KUKA KRL program: MyProgram_040().src

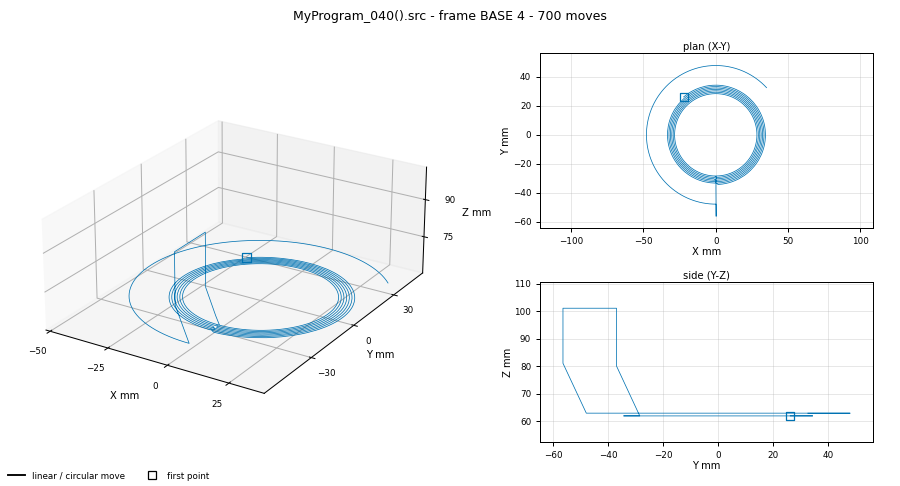
[picture p0: tool path of MyProgram_040().src in frame BASE 4, 700 of 700 moves have a stored position in this frame; points joined in program order, loops and branches not executed]
&ACCESS RVP
&REL 1
&PARAM TEMPLATE = C:\KRC\Roboter\Template\vorgabe
&PARAM EDITMASK = *
DEF MyProgram_040()
; ---- Setting reference (Base) ----
$BASE = BASE_DATA[4]

; --------------------------
; ---- Setting tool (TCP) ----
$TOOL = TOOL_DATA[3]
; --------------------------

$VEL.CP = VEL_APROX_PRINT
Startdeposition()
$VEL.CP = VEL_PRINT
LIN {X -22.2135,Y 26.2071,Z 62,A 121.4467,B 24.8242,C -3.0577,E1 24.9,E2 -758.4485} C_DIS
LIN {X -19.0591,Y 28.5827,Z 62,A 115.8795,B 24.8216,C -3.0802,E1 24.9125,E2 -752.9155} C_DIS
LIN {X -17.4873,Y 29.5709,Z 62,A 112.412,B 24.8214,C -3.0822,E1 24.9208,E2 -749.4421} C_DIS
LIN {X -15.634,Y 30.5912,Z 62,A 108.9316,B 24.8207,C -3.0885,E1 24.9293,E2 -745.967} C_DIS
LIN {X -13.2901,Y 31.6799,Z 62,A 103.9982,B 24.8207,C -3.0886,E1 24.942,E2 -741.0221} C_DIS
LIN {X -10.8187,Y 32.6071,Z 62,A 99.9719,B 24.8196,C -3.0977,E1 24.9525,E2 -737.0096} C_DIS
LIN {X -8.4739,Y 33.2931,Z 62,A 96.4896,B 24.8184,C -3.1079,E1 24.9618,E2 -733.5462} C_DIS
LIN {X -7.1425,Y 33.6045,Z 62,A 93.5529,B 24.819,C -3.1031,E1 24.9699,E2 -730.5943} C_DIS
LIN {X -4.6609,Y 34.0375,Z 62,A 89.325,B 24.8187,C -3.1056,E1 24.9816,E2 -726.3687} C_DIS
LIN {X -2.445,Y 34.2678,Z 62,A 85.3655,B 24.8187,C -3.1047,E1 24.9926,E2 -722.4051} C_DIS
LIN {X 0.711,Y 34.3473,Z 62,A 80.7474,B 24.8178,C -3.1129,E1 25.0054,E2 -717.8067} C_DIS
LIN {X 2.5788,Y 34.2575,Z 62,A 77.4409,B 24.8181,C -3.1108,E1 25.0146,E2 -714.4965} C_DIS
LIN {X 4.6969,Y 34.0324,Z 62,A 74.1424,B 24.8178,C -3.1131,E1 25.0238,E2 -711.2059} C_DIS
LIN {X 6.978,Y 33.6386,Z 62,A 70.5125,B 24.8176,C -3.1144,E1 25.0337,E2 -707.583} C_DIS
LIN {X 8.415,Y 33.3079,Z 62,A 67.7146,B 24.8183,C -3.109,E1 25.0413,E2 -704.7764} C_DIS
LIN {X 10.1674,Y 32.8156,Z 62,A 64.7507,B 24.8184,C -3.1078,E1 25.0493,E2 -701.8147} C_DIS
LIN {X 12.5471,Y 31.9815,Z 62,A 59.7382,B 24.82,C -3.0942,E1 25.0625,E2 -696.7805} C_DIS
LIN {X 14.5005,Y 31.1445,Z 62,A 56.4765,B 24.82,C -3.0937,E1 25.0707,E2 -693.5258} C_DIS
LIN {X 16.8742,Y 29.9253,Z 62,A 52.3714,B 24.8202,C -3.0922,E1 25.0808,E2 -689.4289} C_DIS
LIN {X 19.1187,Y 28.5434,Z 62,A 47.4262,B 24.8218,C -3.0785,E1 25.0924,E2 -684.4673} C_DIS
LIN {X 20.7359,Y 27.3913,Z 62,A 43.8567,B 24.8229,C -3.0695,E1 25.1004,E2 -680.8892} C_DIS
LIN {X 23.4463,Y 25.1103,Z 62,A 38.3676,B 24.8236,C -3.0636,E1 25.1119,E2 -675.408} C_DIS
LIN {X 25.8911,Y 22.5808,Z 62,A 32.7892,B 24.8246,C -3.0549,E1 25.1224,E2 -669.8333} C_DIS
LIN {X 27.3559,Y 20.7829,Z 62,A 29.4122,B 24.8248,C -3.0525,E1 25.1283,E2 -666.4667} C_DIS
LIN {X 28.1113,Y 19.7485,Z 62,A 27.0275,B 24.8258,C -3.0439,E1 25.1322,E2 -664.0731} C_DIS
LIN {X 29.1969,Y 18.1051,Z 62,A 23.9145,B 24.8265,C -3.038,E1 25.1369,E2 -660.9619} C_DIS
LIN {X 30.04,Y 16.6688,Z 62,A 21.2563,B 24.8271,C -3.0324,E1 25.1405,E2 -658.3041} C_DIS
LIN {X 30.6921,Y 15.435,Z 62,A 18.4558,B 24.8286,C -3.0195,E1 25.1441,E2 -655.4879} C_DIS
LIN {X 31.6221,Y 13.4275,Z 62,A 14.5033,B 24.8302,C -3.0056,E1 25.1486,E2 -651.524} C_DIS
LIN {X 32.6254,Y 10.7638,Z 62,A 10.1437,B 24.8311,C -2.9974,E1 25.1526,E2 -647.1695} C_DIS
LIN {X 33.1185,Y 9.1348,Z 62,A 7.3906,B 24.8319,C -2.9902,E1 25.1547,E2 -644.4151} C_DIS
LIN {X 33.5819,Y 7.246,Z 62,A 4.3845,B 24.8327,C -2.9839,E1 25.1566,E2 -641.4115} C_DIS
LIN {X 33.9043,Y 5.5446,Z 62,A 1.3815,B 24.8338,C -2.9735,E1 25.158,E2 -638.4014} C_DIS
LIN {X 34.175,Y 3.5099,Z 62,A -2.0165,B 24.835,C -2.9633,E1 25.1592,E2 -634.9993} C_DIS
LIN {X 34.3202,Y 1.5388,Z 62,A -5.2617,B 24.836,C -2.9538,E1 25.1597,E2 -631.7509} C_DIS
LIN {X 34.3541,Y 0.1987,Z 62,A -7.6725,B 24.8371,C -2.9442,E1 25.1597,E2 -629.3319} C_DIS
LIN {X 34.309,Y -1.7741,Z 62,A -10.9313,B 24.8382,C -2.9344,E1 25.1594,E2 -626.0691} C_DIS
LIN {X 34.0961,Y -4.2062,Z 62,A -14.637,B 24.839,C -2.9269,E1 25.1584,E2 -622.3678} C_DIS
LIN {X 33.8382,Y -5.9366,Z 62,A -17.6519,B 24.8402,C -2.9164,E1 25.157,E2 -619.3456} C_DIS
LIN {X 33.4085,Y -8.0083,Z 62,A -21.3611,B 24.8417,C -2.9028,E1 25.1547,E2 -615.6259} C_DIS
LIN {X 32.8832,Y -9.9486,Z 62,A -24.8083,B 24.8429,C -2.8912,E1 25.152,E2 -612.1708} C_DIS
LIN {X 32.0411,Y -12.3943,Z 62,A -28.5367,B 24.8434,C -2.8866,E1 25.1485,E2 -608.4525} C_DIS
LIN {X 31.434,Y -13.8624,Z 62,A -32.1813,B 24.8458,C -2.8645,E1 25.1444,E2 -604.7755} C_DIS
LIN {X 29.7344,Y -17.2082,Z 62,A -37.2411,B 24.8459,C -2.8637,E1 25.1379,E2 -599.7404} C_DIS
LIN {X 28.506,Y -19.1745,Z 62,A -42.1252,B 24.8486,C -2.8387,E1 25.1304,E2 -594.8215} C_DIS
LIN {X 26.7916,Y -21.5054,Z 62,A -47.2958,B 24.8505,C -2.8213,E1 25.1215,E2 -589.6341} C_DIS
LIN {X 23.923,Y -24.6562,Z 62,A -53.4408,B 24.8509,C -2.8174,E1 25.1097,E2 -583.5064} C_DIS
LIN {X 21.6339,Y -26.6874,Z 62,A -59.2704,B 24.8531,C -2.7963,E1 25.0972,E2 -577.6496} C_DIS
LIN {X 19.7191,Y -28.1322,Z 62,A -63.5381,B 24.8543,C -2.7848,E1 25.0875,E2 -573.3694} C_DIS
LIN {X 15.9551,Y -30.425,Z 62,A -69.5933,B 24.8539,C -2.7889,E1 25.0729,E2 -567.3422} C_DIS
LIN {X 13.6297,Y -31.5353,Z 62,A -74.5651,B 24.8555,C -2.7737,E1 25.0602,E2 -562.3468} C_DIS
LIN {X 11.1987,Y -32.4787,Z 62,A -78.4482,B 24.8555,C -2.774,E1 25.05,E2 -558.4725} C_DIS
LIN {X 9.155,Y -33.1128,Z 62,A -82.0156,B 24.8559,C -2.7701,E1 25.0405,E2 -554.9019} C_DIS
LIN {X 6.777,Y -33.6799,Z 62,A -86.4571,B 24.8567,C -2.762,E1 25.0283,E2 -550.447} C_DIS
LIN {X 4.3543,Y -34.0777,Z 62,A -89.9455,B 24.8562,C -2.7665,E1 25.0187,E2 -546.9726} C_DIS
LIN {X 1.6468,Y -34.3153,Z 62,A -95.2543,B 24.8574,C -2.7554,E1 25.0039,E2 -541.6397} C_DIS
LIN {X 1.6468,Y -34.3153,Z 62,A -95.2543,B 24.8574,C -2.7554,E1 25.0039,E2 -541.6397} C_DIS
Enddeposition()
LIN {X 0.1829,Y -33.3699,Z 62,A -96.4469,B 24.8542,C -2.7864,E1 25.0008,E2 -540.5209} C_DIS
Startdeposition()
$VEL.CP = VEL_PRINT
LIN {X 1.4228,Y -33.3445,Z 62,A -93.237,B 24.8528,C -2.7995,E1 25.0098,E2 -543.7614} C_DIS
LIN {X 3.8682,Y -33.1501,Z 62,A -89.4536,B 24.8531,C -2.7966,E1 25.0203,E2 -547.5356} C_DIS
LIN {X 6.4667,Y -32.7422,Z 62,A -84.1849,B 24.8518,C -2.8092,E1 25.0348,E2 -552.8286} C_DIS
LIN {X 8.6813,Y -32.2262,Z 62,A -80.8923,B 24.8521,C -2.8055,E1 25.0437,E2 -556.1074} C_DIS
LIN {X 10.7356,Y -31.6013,Z 62,A -76.8197,B 24.8512,C -2.8147,E1 25.0546,E2 -560.1942} C_DIS
LIN {X 13.1904,Y -30.658,Z 62,A -72.1573,B 24.8503,C -2.8228,E1 25.0667,E2 -564.8654} C_DIS
LIN {X 15.1524,Y -29.7371,Z 62,A -69.1058,B 24.8506,C -2.82,E1 25.0743,E2 -567.9021} C_DIS
LIN {X 16.9825,Y -28.7313,Z 62,A -64.8683,B 24.849,C -2.8349,E1 25.0846,E2 -572.1622} C_DIS
LIN {X 18.9767,Y -27.4551,Z 62,A -61.3792,B 24.849,C -2.8349,E1 25.0927,E2 -575.6399} C_DIS
LIN {X 21.2128,Y -25.7669,Z 62,A -55.8058,B 24.8468,C -2.8555,E1 25.105,E2 -581.2413} C_DIS
LIN {X 22.9178,Y -24.2625,Z 62,A -51.6212,B 24.8454,C -2.8684,E1 25.1135,E2 -585.4392} C_DIS
LIN {X 25.8376,Y -21.1265,Z 62,A -45.1587,B 24.8448,C -2.8741,E1 25.1255,E2 -591.8865} C_DIS
LIN {X 27.6388,Y -18.708,Z 62,A -39.68,B 24.8428,C -2.8922,E1 25.1344,E2 -597.3815} C_DIS
LIN {X 29.0319,Y -16.4634,Z 62,A -35.1975,B 24.8415,C -2.9042,E1 25.1408,E2 -601.8693} C_DIS
LIN {X 30.4402,Y -13.6854,Z 62,A -30.0332,B 24.8401,C -2.9171,E1 25.147,E2 -607.0365} C_DIS
LIN {X 31.2986,Y -11.588,Z 62,A -26.4051,B 24.8392,C -2.925,E1 25.1507,E2 -610.6631} C_DIS
LIN {X 31.92,Y -9.7482,Z 62,A -22.6045,B 24.8374,C -2.9419,E1 25.1539,E2 -614.4821} C_DIS
LIN {X 32.7265,Y -6.5492,Z 62,A -17.7367,B 24.8367,C -2.9479,E1 25.157,E2 -619.3359} C_DIS
LIN {X 32.9464,Y -5.3344,Z 62,A -14.5179,B 24.8342,C -2.9705,E1 25.1584,E2 -622.5894} C_DIS
LIN {X 33.3383,Y -1.5702,Z 62,A -9.092,B 24.8336,C -2.9753,E1 25.1597,E2 -627.9943} C_DIS
LIN {X 33.375,Y 0.0538,Z 62,A -6.2185,B 24.8325,C -2.9852,E1 25.1597,E2 -630.8742} C_DIS
LIN {X 33.3259,Y 1.8094,Z 62,A -3.2231,B 24.8315,C -2.9943,E1 25.1594,E2 -633.8734} C_DIS
LIN {X 33.2052,Y 3.364,Z 62,A -0.7318,B 24.8308,C -2.9999,E1 25.1588,E2 -636.3632} C_DIS
LIN {X 33.0427,Y 4.6979,Z 62,A 1.6423,B 24.8299,C -3.008,E1 25.1579,E2 -638.7425} C_DIS
LIN {X 32.7913,Y 6.2155,Z 62,A 4.524,B 24.8286,C -3.0195,E1 25.1565,E2 -641.6345} C_DIS
LIN {X 32.2699,Y 8.5188,Z 62,A 8.4206,B 24.8275,C -3.0294,E1 25.1539,E2 -645.5319} C_DIS
LIN {X 31.633,Y 10.6416,Z 62,A 12.4439,B 24.8259,C -3.0436,E1 25.1505,E2 -649.566} C_DIS
LIN {X 30.8002,Y 12.855,Z 62,A 16.3295,B 24.8248,C -3.0526,E1 25.1465,E2 -653.4515} C_DIS
LIN {X 29.4508,Y 15.7026,Z 62,A 22.0288,B 24.8227,C -3.0713,E1 25.1394,E2 -659.1647} C_DIS
LIN {X 28.245,Y 17.7799,Z 62,A 25.5541,B 24.8224,C -3.0736,E1 25.1343,E2 -662.6774} C_DIS
LIN {X 27.4035,Y 19.051,Z 62,A 28.1395,B 24.8217,C -3.0796,E1 25.1303,E2 -665.2643} C_DIS
LIN {X 26.5171,Y 20.267,Z 62,A 30.6298,B 24.8211,C -3.0845,E1 25.1261,E2 -667.7543} C_DIS
LIN {X 25.6944,Y 21.3,Z 62,A 32.9585,B 24.8204,C -3.0906,E1 25.122,E2 -670.0865} C_DIS
LIN {X 24.7958,Y 22.3399,Z 62,A 36.0169,B 24.8187,C -3.1052,E1 25.1163,E2 -673.1659} C_DIS
LIN {X 22.7484,Y 24.4218,Z 62,A 40.7734,B 24.8179,C -3.1119,E1 25.1067,E2 -677.9187} C_DIS
LIN {X 20.6615,Y 26.2106,Z 62,A 45.0491,B 24.8176,C -3.1148,E1 25.0976,E2 -682.1848} C_DIS
LIN {X 19.1465,Y 27.337,Z 62,A 48.6346,B 24.8164,C -3.1247,E1 25.0894,E2 -685.7811} C_DIS
LIN {X 17.0397,Y 28.6975,Z 62,A 52.5144,B 24.8164,C -3.1256,E1 25.0803,E2 -689.6509} C_DIS
LIN {X 15.4263,Y 29.5963,Z 62,A 55.9993,B 24.8154,C -3.1337,E1 25.0717,E2 -693.145} C_DIS
LIN {X 13.597,Y 30.48,Z 62,A 59.7045,B 24.8146,C -3.1404,E1 25.0623,E2 -696.8566} C_DIS
LIN {X 11.4187,Y 31.3607,Z 62,A 63.0646,B 24.8151,C -3.136,E1 25.0536,E2 -700.199} C_DIS
LIN {X 10.1374,Y 31.7985,Z 62,A 65.3843,B 24.8149,C -3.1378,E1 25.0474,E2 -702.5184} C_DIS
LIN {X 8.378,Y 32.3064,Z 62,A 68.9747,B 24.814,C -3.1451,E1 25.0377,E2 -706.1203} C_DIS
LIN {X 6.1328,Y 32.8069,Z 62,A 72.6936,B 24.8141,C -3.1441,E1 25.0276,E2 -709.8324} C_DIS
LIN {X 4.5023,Y 33.0705,Z 62,A 75.876,B 24.8136,C -3.1488,E1 25.0187,E2 -713.0232} C_DIS
LIN {X 1.7164,Y 33.3311,Z 62,A 81.564,B 24.8124,C -3.1589,E1 25.0028,E2 -718.7328} C_DIS
LIN {X -2.4774,Y 33.2834,Z 62,A 87.3966,B 24.8144,C -3.1417,E1 24.9867,E2 -724.5252} C_DIS
LIN {X -3.8653,Y 33.1504,Z 62,A 90.0327,B 24.8142,C -3.143,E1 24.9793,E2 -727.1661} C_DIS
LIN {X -5.6675,Y 32.8906,Z 62,A 93.1198,B 24.8146,C -3.1405,E1 24.9708,E2 -730.25} C_DIS
LIN {X -7.3587,Y 32.554,Z 62,A 96.5725,B 24.8142,C -3.1431,E1 24.9614,E2 -733.7131} C_DIS
LIN {X -9.9318,Y 31.8625,Z 62,A 100.6041,B 24.8155,C -3.1328,E1 24.9506,E2 -737.7267} C_DIS
LIN {X -12.8323,Y 30.8096,Z 62,A 106.8089,B 24.8152,C -3.1348,E1 24.9344,E2 -743.9496} C_DIS
LIN {X -15.1762,Y 29.725,Z 62,A 110.2748,B 24.8171,C -3.1186,E1 24.9258,E2 -747.3857} C_DIS
LIN {X -16.7138,Y 28.8886,Z 62,A 113.5931,B 24.8174,C -3.1165,E1 24.9177,E2 -750.7086} C_DIS
LIN {X -18.3349,Y 27.8877,Z 62,A 117.4181,B 24.8174,C -3.1156,E1 24.9087,E2 -754.5439} C_DIS
LIN {X -21.0824,Y 25.8722,Z 62,A 122.2135,B 24.82,C -3.094,E1 24.8981,E2 -759.305} C_DIS
LIN {X -22.0783,Y 25.0293,Z 62,A 126.1085,B 24.8189,C -3.104,E1 24.8899,E2 -763.2393} C_DIS
LIN {X -25.5295,Y 21.4982,Z 62,A 134.6867,B 24.8212,C -3.0841,E1 24.8738,E2 -771.808} C_DIS
LIN {X -28.2172,Y 17.8241,Z 62,A 141.0536,B 24.825,C -3.0507,E1 24.8638,E2 -778.1262} C_DIS
LIN {X -28.9128,Y 16.6716,Z 62,A 143.5735,B 24.8256,C -3.046,E1 24.8602,E2 -780.648} C_DIS
LIN {X -29.7714,Y 15.0848,Z 62,A 146.4195,B 24.8268,C -3.0351,E1 24.8565,E2 -783.4829} C_DIS
LIN {X -30.2718,Y 14.0538,Z 62,A 149.4607,B 24.8265,C -3.0383,E1 24.8529,E2 -786.5483} C_DIS
LIN {X -31.6705,Y 10.5303,Z 62,A 154.8201,B 24.8298,C -3.0093,E1 24.8477,E2 -791.8686} C_DIS
LIN {X -32.3711,Y 8.1254,Z 62,A 160.5197,B 24.83,C -3.0075,E1 24.8435,E2 -797.5971} C_DIS
LIN {X -32.8497,Y 5.8982,Z 62,A 164.193,B 24.8316,C -2.9934,E1 24.8416,E2 -801.2584} C_DIS
LIN {X -33.2606,Y 2.7623,Z 62,A 169.0956,B 24.834,C -2.9722,E1 24.8401,E2 -806.1394} C_DIS
LIN {X -33.3722,Y 0.439,Z 62,A 173.4965,B 24.835,C -2.963,E1 24.8398,E2 -810.5449} C_DIS
LIN {X -33.3243,Y -1.8394,Z 62,A 177.3186,B 24.8364,C -2.9501,E1 24.8402,E2 -814.359} C_DIS
LIN {X -33.1418,Y -3.9387,Z 62,A -179.5093,B 24.8381,C -2.9353,E1 24.8411,E2 -817.5147} C_DIS
LIN {X -32.9043,Y -5.5852,Z 62,A -176.45,B 24.8389,C -2.9282,E1 24.8425,E2 -820.5753} C_DIS
LIN {X -32.5254,Y -7.4827,Z 62,A -173.0592,B 24.8399,C -2.9188,E1 24.8445,E2 -823.9635} C_DIS
LIN {X -31.9568,Y -9.6266,Z 62,A -169.2266,B 24.8411,C -2.9078,E1 24.8474,E2 -827.7919} C_DIS
LIN {X -31.1362,Y -12.0183,Z 62,A -164.5872,B 24.8422,C -2.8979,E1 24.8518,E2 -832.4338} C_DIS
LIN {X -30.1887,Y -14.2317,Z 62,A -160.582,B 24.8436,C -2.8854,E1 24.8564,E2 -836.4311} C_DIS
LIN {X -29.4655,Y -15.6747,Z 62,A -157.8731,B 24.8444,C -2.8774,E1 24.8599,E2 -839.1354} C_DIS
LIN {X -28.295,Y -17.6999,Z 62,A -153.9787,B 24.8457,C -2.8661,E1 24.8655,E2 -843.0228} C_DIS
LIN {X -27.374,Y -19.0935,Z 62,A -151.2935,B 24.8466,C -2.8574,E1 24.8697,E2 -845.7005} C_DIS
LIN {X -26.456,Y -20.3464,Z 62,A -148.4701,B 24.8471,C -2.8525,E1 24.8744,E2 -848.5257} C_DIS
LIN {X -25.3348,Y -21.7268,Z 62,A -145.3707,B 24.8478,C -2.846,E1 24.88,E2 -851.6239} C_DIS
LIN {X -24.0752,Y -23.1145,Z 62,A -142.0378,B 24.8485,C -2.8402,E1 24.8863,E2 -854.9575} C_DIS
LIN {X -22.8098,Y -24.3641,Z 62,A -139.1432,B 24.8493,C -2.8326,E1 24.8921,E2 -857.8459} C_DIS
LIN {X -21.4959,Y -25.5315,Z 62,A -135.9256,B 24.8497,C -2.8288,E1 24.8989,E2 -861.0671} C_DIS
LIN {X -20.1533,Y -26.6033,Z 62,A -133.0951,B 24.8503,C -2.8226,E1 24.9052,E2 -863.893} C_DIS
LIN {X -19.0218,Y -27.4238,Z 62,A -130.6625,B 24.8507,C -2.819,E1 24.9107,E2 -866.3255} C_DIS
LIN {X -17.5805,Y -28.3691,Z 62,A -127.8621,B 24.8513,C -2.813,E1 24.9173,E2 -869.1206} C_DIS
LIN {X -16.4044,Y -29.0655,Z 62,A -124.8197,B 24.8509,C -2.8168,E1 24.9247,E2 -872.181} C_DIS
LIN {X -13.5755,Y -30.4886,Z 62,A -119.851,B 24.8521,C -2.8058,E1 24.9372,E2 -877.1361} C_DIS
LIN {X -11.4437,Y -31.3518,Z 62,A -115.6595,B 24.8522,C -2.8047,E1 24.9481,E2 -881.334} C_DIS
LIN {X -9.364,Y -32.0344,Z 62,A -112.1793,B 24.8528,C -2.7991,E1 24.9574,E2 -884.8067} C_DIS
LIN {X -7.588,Y -32.5011,Z 62,A -109.002,B 24.853,C -2.7976,E1 24.966,E2 -887.9851} C_DIS
LIN {X -5.2723,Y -32.9563,Z 62,A -105.3031,B 24.8535,C -2.7924,E1 24.9761,E2 -891.6754} C_DIS
LIN {X -3.9275,Y -33.1431,Z 62,A -102.0223,B 24.8524,C -2.8027,E1 24.9853,E2 -894.983} C_DIS
LIN {X -0.4827,Y -33.3718,Z 62,A -96.4764,B 24.8529,C -2.7988,E1 25.0008,E2 -900.5209} C_DIS
LIN {X -0.4827,Y -33.3718,Z 62,A -96.4764,B 24.8529,C -2.7988,E1 25.0008,E2 -900.5209} C_DIS
Enddeposition()
LIN {X 0.1538,Y -32.3933,Z 62,A -94.978,B 24.8506,C -2.8203,E1 25.0051,E2 -902.0704} C_DIS
Startdeposition()
$VEL.CP = VEL_PRINT
LIN {X -0.5076,Y -32.3915,Z 62,A -99.0735,B 24.854,C -2.7876,E1 24.9934,E2 -897.897} C_DIS
LIN {X -4.373,Y -32.0994,Z 62,A -105.0397,B 24.853,C -2.7975,E1 24.9769,E2 -891.9514} C_DIS
LIN {X -6.3091,Y -31.7751,Z 62,A -108.8338,B 24.8532,C -2.7954,E1 24.9665,E2 -888.1481} C_DIS
LIN {X -7.9655,Y -31.401,Z 62,A -111.4444,B 24.8526,C -2.8009,E1 24.9594,E2 -885.5472} C_DIS
LIN {X -9.3688,Y -31.0112,Z 62,A -114.1241,B 24.8526,C -2.8015,E1 24.9522,E2 -882.8646} C_DIS
LIN {X -11.1696,Y -30.409,Z 62,A -117.88,B 24.8526,C -2.8004,E1 24.9423,E2 -879.0986} C_DIS
LIN {X -13.109,Y -29.6245,Z 62,A -121.8566,B 24.8526,C -2.8015,E1 24.9321,E2 -875.1154} C_DIS
LIN {X -15.677,Y -28.3497,Z 62,A -126.6654,B 24.8516,C -2.8103,E1 24.9202,E2 -870.3145} C_DIS
LIN {X -17.8366,Y -27.0428,Z 62,A -131.0512,B 24.8509,C -2.8176,E1 24.9098,E2 -865.9322} C_DIS
LIN {X -19.3899,Y -25.9517,Z 62,A -134.7425,B 24.8506,C -2.8202,E1 24.9015,E2 -862.2341} C_DIS
LIN {X -21.5251,Y -24.2103,Z 62,A -139.2977,B 24.8493,C -2.832,E1 24.8918,E2 -857.6895} C_DIS
LIN {X -23.1553,Y -22.6552,Z 62,A -142.8697,B 24.8481,C -2.8437,E1 24.8847,E2 -854.1304} C_DIS
LIN {X -24.03,Y -21.7266,Z 62,A -145.2172,B 24.8476,C -2.8477,E1 24.8803,E2 -851.7822} C_DIS
LIN {X -24.829,Y -20.8079,Z 62,A -147.7786,B 24.8475,C -2.8491,E1 24.8756,E2 -849.2125} C_DIS
LIN {X -26.2704,Y -18.9567,Z 62,A -151.6984,B 24.8462,C -2.8608,E1 24.869,E2 -845.3018} C_DIS
LIN {X -27.3955,Y -17.2906,Z 62,A -155.6893,B 24.8457,C -2.8662,E1 24.8629,E2 -841.3037} C_DIS
LIN {X -28.4065,Y -15.5742,Z 62,A -159.6717,B 24.845,C -2.8718,E1 24.8575,E2 -837.3138} C_DIS
LIN {X -29.8675,Y -12.5455,Z 62,A -164.8424,B 24.8426,C -2.8942,E1 24.8515,E2 -832.1685} C_DIS
LIN {X -30.5226,Y -10.8549,Z 62,A -168.2138,B 24.8417,C -2.9021,E1 24.8483,E2 -828.7969} C_DIS
LIN {X -31.1641,Y -8.8464,Z 62,A -171.7727,B 24.8404,C -2.9143,E1 24.8454,E2 -825.2468} C_DIS
LIN {X -31.5598,Y -7.3102,Z 62,A -174.967,B 24.8398,C -2.9197,E1 24.8433,E2 -822.0467} C_DIS
LIN {X -32.0757,Y -4.5397,Z 62,A -179.2334,B 24.8375,C -2.9403,E1 24.8413,E2 -817.8044} C_DIS
LIN {X -32.3364,Y -1.9611,Z 62,A 175.4432,B 24.8366,C -2.9489,E1 24.8399,E2 -812.4696} C_DIS
LIN {X -32.3954,Y -0.0822,Z 62,A 172.3891,B 24.8352,C -2.9613,E1 24.8398,E2 -809.4268} C_DIS
LIN {X -32.3655,Y 1.3908,Z 62,A 169.7508,B 24.8343,C -2.9692,E1 24.84,E2 -806.7915} C_DIS
LIN {X -32.2529,Y 3.0349,Z 62,A 166.6061,B 24.8335,C -2.9766,E1 24.8408,E2 -803.6457} C_DIS
LIN {X -31.9024,Y 5.6309,Z 62,A 162.6508,B 24.8313,C -2.9962,E1 24.8423,E2 -799.7135} C_DIS
LIN {X -31.4815,Y 7.6404,Z 62,A 157.9411,B 24.8309,C -2.9993,E1 24.8452,E2 -794.9837} C_DIS
LIN {X -30.8287,Y 9.9525,Z 62,A 153.8984,B 24.8293,C -3.0138,E1 24.8485,E2 -790.9524} C_DIS
LIN {X -30.0364,Y 12.1339,Z 62,A 150.0939,B 24.8276,C -3.0283,E1 24.8522,E2 -787.1613} C_DIS
LIN {X -29.2829,Y 13.8567,Z 62,A 146.563,B 24.8267,C -3.0365,E1 24.8563,E2 -783.6306} C_DIS
LIN {X -28.667,Y 15.0882,Z 62,A 143.6364,B 24.8263,C -3.0397,E1 24.8601,E2 -780.6962} C_DIS
LIN {X -27.1784,Y 17.6297,Z 62,A 138.4491,B 24.8246,C -3.0543,E1 24.8677,E2 -775.5171} C_DIS
LIN {X -25.3386,Y 20.1849,Z 62,A 133.5089,B 24.8224,C -3.0738,E1 24.8759,E2 -770.5999} C_DIS
LIN {X -24.417,Y 21.2901,Z 62,A 130.0547,B 24.8224,C -3.0729,E1 24.8823,E2 -767.1279} C_DIS
LIN {X -21.8354,Y 23.9308,Z 62,A 124.1905,B 24.8201,C -3.0935,E1 24.8939,E2 -761.2885} C_DIS
LIN {X -20.881,Y 24.7676,Z 62,A 121.1991,B 24.8202,C -3.0922,E1 24.9004,E2 -758.2823} C_DIS
LIN {X -18.1589,Y 26.8275,Z 62,A 115.7342,B 24.8183,C -3.109,E1 24.9127,E2 -752.8386} C_DIS
LIN {X -16.1624,Y 28.0755,Z 62,A 112.0613,B 24.8169,C -3.1208,E1 24.9214,E2 -749.1825} C_DIS
LIN {X -14.7245,Y 28.8556,Z 62,A 109.2787,B 24.8162,C -3.1265,E1 24.9282,E2 -746.4058} C_DIS
LIN {X -12.9577,Y 29.691,Z 62,A 104.8369,B 24.8167,C -3.1226,E1 24.9396,E2 -741.9439} C_DIS
LIN {X -11.0027,Y 30.4698,Z 62,A 101.8142,B 24.8153,C -3.1339,E1 24.9474,E2 -738.9417} C_DIS
LIN {X -9.8011,Y 30.8777,Z 62,A 99.6031,B 24.815,C -3.1368,E1 24.9533,E2 -736.7335} C_DIS
LIN {X -7.687,Y 31.4701,Z 62,A 95.3806,B 24.815,C -3.1374,E1 24.9647,E2 -732.5061} C_DIS
LIN {X -5.4538,Y 31.9332,Z 62,A 91.4709,B 24.8144,C -3.1417,E1 24.9754,E2 -728.6025} C_DIS
LIN {X -3.8013,Y 32.1716,Z 62,A 88.5536,B 24.8142,C -3.1439,E1 24.9834,E2 -725.688} C_DIS
LIN {X -2.2721,Y 32.3157,Z 62,A 85.5132,B 24.8144,C -3.1418,E1 24.9919,E2 -722.6414} C_DIS
LIN {X 0.5244,Y 32.3912,Z 62,A 80.6379,B 24.8142,C -3.1436,E1 25.0055,E2 -717.7703} C_DIS
LIN {X 2.6938,Y 32.2831,Z 62,A 77.0702,B 24.8138,C -3.1465,E1 25.0154,E2 -714.211} C_DIS
LIN {X 4.3107,Y 32.1076,Z 62,A 74.0143,B 24.8141,C -3.144,E1 25.0239,E2 -711.1516} C_DIS
LIN {X 6.2253,Y 31.7916,Z 62,A 70.728,B 24.8141,C -3.1444,E1 25.0329,E2 -707.8697} C_DIS
LIN {X 8.1548,Y 31.3523,Z 62,A 66.8724,B 24.8148,C -3.1385,E1 25.0434,E2 -704.0058} C_DIS
LIN {X 10.0774,Y 30.7883,Z 62,A 63.5437,B 24.8148,C -3.1383,E1 25.0523,E2 -700.6826} C_DIS
LIN {X 11.9753,Y 30.1006,Z 62,A 59.8961,B 24.8153,C -3.1341,E1 25.0618,E2 -697.0329} C_DIS
LIN {X 13.9209,Y 29.252,Z 62,A 56.3645,B 24.8155,C -3.1325,E1 25.0708,E2 -693.5063} C_DIS
LIN {X 15.2443,Y 28.5847,Z 62,A 53.8398,B 24.8158,C -3.1303,E1 25.077,E2 -690.9835} C_DIS
LIN {X 16.3177,Y 27.9861,Z 62,A 51.5537,B 24.8163,C -3.126,E1 25.0826,E2 -688.6938} C_DIS
LIN {X 17.6959,Y 27.1343,Z 62,A 48.6532,B 24.8168,C -3.1212,E1 25.0894,E2 -685.7916} C_DIS
LIN {X 19.3257,Y 26.0001,Z 62,A 45.3473,B 24.8172,C -3.1179,E1 25.0969,E2 -682.4893} C_DIS
LIN {X 20.4469,Y 25.1274,Z 62,A 42.5184,B 24.8182,C -3.1095,E1 25.1031,E2 -679.651} C_DIS
LIN {X 22.0505,Y 23.7334,Z 62,A 38.7589,B 24.8191,C -3.1022,E1 25.1109,E2 -675.8892} C_DIS
LIN {X 23.6533,Y 22.135,Z 62,A 35.2331,B 24.8193,C -3.0999,E1 25.1178,E2 -672.3731} C_DIS
LIN {X 24.5119,Y 21.1814,Z 62,A 32.8349,B 24.8201,C -3.0932,E1 25.1222,E2 -669.9698} C_DIS
LIN {X 25.6781,Y 19.7509,Z 62,A 29.4461,B 24.8212,C -3.084,E1 25.1281,E2 -666.575} C_DIS
LIN {X 26.6952,Y 18.3531,Z 62,A 26.2572,B 24.8223,C -3.0748,E1 25.1332,E2 -663.3799} C_DIS
LIN {X 27.7387,Y 16.7343,Z 62,A 23.0323,B 24.823,C -3.0686,E1 25.138,E2 -660.1565} C_DIS
LIN {X 28.5766,Y 15.2594,Z 62,A 19.1467,B 24.8253,C -3.0489,E1 25.1432,E2 -656.2447} C_DIS
LIN {X 29.8737,Y 12.5308,Z 62,A 14.7774,B 24.8255,C -3.0471,E1 25.1482,E2 -651.8949} C_DIS
LIN {X 30.7022,Y 10.336,Z 62,A 9.96,B 24.8279,C -3.0262,E1 25.1527,E2 -647.0549} C_DIS
LIN {X 31.4172,Y 7.9012,Z 62,A 6.1636,B 24.8283,C -3.0223,E1 25.1555,E2 -643.2711} C_DIS
LIN {X 31.8546,Y 5.8966,Z 62,A 2.396,B 24.8298,C -3.0094,E1 25.1576,E2 -639.495} C_DIS
LIN {X 32.1672,Y 3.8374,Z 62,A -1.1222,B 24.8308,C -3.0004,E1 25.1589,E2 -635.9762} C_DIS
LIN {X 32.3286,Y 2.0807,Z 62,A -4.6979,B 24.8326,C -2.9844,E1 25.1596,E2 -632.3839} C_DIS
LIN {X 32.3757,Y -1.1372,Z 62,A -10.0928,B 24.8341,C -2.9707,E1 25.1596,E2 -626.9887} C_DIS
LIN {X 32.2483,Y -3.0813,Z 62,A -13.1917,B 24.8348,C -2.9647,E1 25.1589,E2 -623.894} C_DIS
LIN {X 31.9751,Y -5.2034,Z 62,A -17.2389,B 24.8365,C -2.9493,E1 25.1572,E2 -619.834} C_DIS
LIN {X 31.3522,Y -8.1542,Z 62,A -22.8001,B 24.8387,C -2.9296,E1 25.1537,E2 -614.2585} C_DIS
LIN {X 30.7613,Y -10.1607,Z 62,A -25.8591,B 24.839,C -2.9272,E1 25.1512,E2 -611.2111} C_DIS
LIN {X 30.0947,Y -11.9894,Z 62,A -30.0232,B 24.8412,C -2.907,E1 25.147,E2 -607.0223} C_DIS
LIN {X 28.8736,Y -14.6894,Z 62,A -34.8647,B 24.8423,C -2.8971,E1 25.1412,E2 -602.1836} C_DIS
LIN {X 27.8924,Y -16.4765,Z 62,A -38.2162,B 24.843,C -2.8904,E1 25.1366,E2 -598.8334} C_DIS
LIN {X 26.9767,Y -17.9365,Z 62,A -41.5971,B 24.8444,C -2.8775,E1 25.1314,E2 -595.439} C_DIS
LIN {X 25.5456,Y -19.9228,Z 62,A -45.8046,B 24.8455,C -2.8677,E1 25.1243,E2 -591.2284} C_DIS
LIN {X 23.4736,Y -22.3253,Z 62,A -51.6807,B 24.8474,C -2.8504,E1 25.1133,E2 -585.3374} C_DIS
LIN {X 21.8548,Y -23.913,Z 62,A -54.9989,B 24.8474,C -2.8501,E1 25.1066,E2 -582.0322} C_DIS
LIN {X 20.6428,Y -24.9668,Z 62,A -58.3004,B 24.8487,C -2.8379,E1 25.0996,E2 -578.7145} C_DIS
LIN {X 18.6695,Y -26.4753,Z 62,A -61.9654,B 24.8487,C -2.8383,E1 25.0914,E2 -575.0635} C_DIS
LIN {X 17.4782,Y -27.2759,Z 62,A -64.7838,B 24.8496,C -2.8299,E1 25.0848,E2 -572.2345} C_DIS
LIN {X 16.1866,Y -28.0616,Z 62,A -67.2912,B 24.8498,C -2.8272,E1 25.0788,E2 -569.7284} C_DIS
LIN {X 14.6704,Y -28.8833,Z 62,A -70.6419,B 24.8508,C -2.8184,E1 25.0704,E2 -566.3662} C_DIS
LIN {X 12.7469,Y -29.7825,Z 62,A -74.4502,B 24.8514,C -2.8121,E1 25.0607,E2 -562.5525} C_DIS
LIN {X 10.2738,Y -30.7232,Z 62,A -79.6833,B 24.8528,C -2.7996,E1 25.0469,E2 -557.3005} C_DIS
LIN {X 7.79,Y -31.445,Z 62,A -83.5535,B 24.8524,C -2.8032,E1 25.0365,E2 -553.4448} C_DIS
LIN {X 5.9267,Y -31.8488,Z 62,A -87.0927,B 24.8529,C -2.7984,E1 25.0268,E2 -549.8985} C_DIS
LIN {X 3.7253,Y -32.1805,Z 62,A -91.678,B 24.8539,C -2.7886,E1 25.0141,E2 -545.2937} C_DIS
LIN {X 0.1538,Y -32.3933,Z 62,A -94.9778,B 24.8506,C -2.8202,E1 25.0051,E2 -542.0704} C_DIS
Enddeposition()
LIN {X 0.1538,Y -32.3933,Z 62,A -94.9778,B 24.8506,C -2.8202,E1 25.0051,E2 -542.0704} C_DIS
Startdeposition()
$VEL.CP = VEL_PRINT
LIN {X 0.7496,Y -31.4064,Z 62,A -94.2132,B 24.8492,C -2.8335,E1 25.0073,E2 -542.8662} C_DIS
LIN {X 3.5993,Y -31.2089,Z 62,A -89.2707,B 24.8492,C -2.833,E1 25.021,E2 -547.8049} C_DIS
LIN {X 5.6125,Y -30.9104,Z 62,A -85.5961,B 24.849,C -2.8353,E1 25.0312,E2 -551.4812} C_DIS
LIN {X 7.6188,Y -30.4784,Z 62,A -82.3726,B 24.8493,C -2.8327,E1 25.0399,E2 -554.6942} C_DIS
LIN {X 9.8387,Y -29.8349,Z 62,A -76.8318,B 24.847,C -2.8533,E1 25.0548,E2 -560.2738} C_DIS
LIN {X 12.2975,Y -28.909,Z 62,A -72.976,B 24.8476,C -2.8485,E1 25.0647,E2 -564.1095} C_DIS
LIN {X 14.0717,Y -28.0878,Z 62,A -68.7808,B 24.8461,C -2.8618,E1 25.0753,E2 -568.3254} C_DIS
LIN {X 16.5071,Y -26.7299,Z 62,A -63.7587,B 24.8452,C -2.8701,E1 25.0874,E2 -573.3517} C_DIS
LIN {X 18.6769,Y -25.2615,Z 62,A -59.3217,B 24.8447,C -2.8752,E1 25.0975,E2 -577.7856} C_DIS
LIN {X 20.0444,Y -24.1903,Z 62,A -55.9443,B 24.8436,C -2.8848,E1 25.1048,E2 -581.1727} C_DIS
LIN {X 21.8114,Y -22.6099,Z 62,A -51.8187,B 24.8428,C -2.8921,E1 25.1133,E2 -585.2989} C_DIS
LIN {X 23.7112,Y -20.6091,Z 62,A -46.9653,B 24.8417,C -2.9021,E1 25.1224,E2 -590.1545} C_DIS
LIN {X 24.9916,Y -19.0367,Z 62,A -43.1573,B 24.8405,C -2.9132,E1 25.129,E2 -593.9708} C_DIS
LIN {X 26.1869,Y -17.355,Z 62,A -40.1154,B 24.8405,C -2.9137,E1 25.1338,E2 -596.999} C_DIS
LIN {X 27.0704,Y -15.9416,Z 62,A -36.4253,B 24.8386,C -2.9309,E1 25.1392,E2 -600.7111} C_DIS
LIN {X 28.001,Y -14.2441,Z 62,A -32.9225,B 24.8375,C -2.9407,E1 25.1438,E2 -604.2186} C_DIS
LIN {X 29.2119,Y -11.5593,Z 62,A -27.0598,B 24.835,C -2.9633,E1 25.1502,E2 -610.1027} C_DIS
LIN {X 29.993,Y -9.3472,Z 62,A -22.7558,B 24.8335,C -2.9767,E1 25.1539,E2 -614.414} C_DIS
LIN {X 30.7209,Y -6.572,Z 62,A -18.15,B 24.8326,C -2.9842,E1 25.1568,E2 -619.0108} C_DIS
LIN {X 31.0905,Y -4.5095,Z 62,A -14.6388,B 24.8318,C -2.9918,E1 25.1584,E2 -622.5195} C_DIS
LIN {X 31.3537,Y -1.9756,Z 62,A -9.9085,B 24.83,C -3.0075,E1 25.1596,E2 -627.2589} C_DIS
LIN {X 31.4045,Y 0.8349,Z 62,A -3.6332,B 24.8263,C -3.0395,E1 25.1595,E2 -633.5727} C_DIS
LIN {X 31.0684,Y 4.6588,Z 62,A 2.3726,B 24.8255,C -3.0472,E1 25.1575,E2 -639.5613} C_DIS
LIN {X 30.7591,Y 6.3896,Z 62,A 5.0493,B 24.8252,C -3.0497,E1 25.1561,E2 -642.2281} C_DIS
LIN {X 30.4607,Y 7.6871,Z 62,A 7.9592,B 24.8236,C -3.0635,E1 25.1542,E2 -645.154} C_DIS
LIN {X 29.8075,Y 9.9234,Z 62,A 12.3362,B 24.8219,C -3.0776,E1 25.1505,E2 -649.5396} C_DIS
LIN {X 28.9651,Y 12.1644,Z 62,A 16.2828,B 24.8212,C -3.0843,E1 25.1465,E2 -653.4801} C_DIS
LIN {X 28.4286,Y 13.3708,Z 62,A 18.5623,B 24.8206,C -3.0892,E1 25.1438,E2 -655.759} C_DIS
LIN {X 27.8327,Y 14.5703,Z 62,A 21.1486,B 24.8196,C -3.0977,E1 25.1405,E2 -658.3516} C_DIS
LIN {X 26.883,Y 16.2559,Z 62,A 24.7038,B 24.8185,C -3.1072,E1 25.1355,E2 -661.9111} C_DIS
LIN {X 25.986,Y 17.6543,Z 62,A 27.8975,B 24.8173,C -3.1169,E1 25.1305,E2 -665.1119} C_DIS
LIN {X 24.6614,Y 19.4619,Z 62,A 31.5013,B 24.8169,C -3.1203,E1 25.1244,E2 -668.7065} C_DIS
LIN {X 23.8129,Y 20.4918,Z 62,A 34.2078,B 24.8159,C -3.1293,E1 25.1195,E2 -671.422} C_DIS
LIN {X 22.4966,Y 21.9276,Z 62,A 37.4837,B 24.8154,C -3.1334,E1 25.1133,E2 -674.6933} C_DIS
LIN {X 21.3523,Y 23.0445,Z 62,A 40.4231,B 24.8147,C -3.1395,E1 25.1073,E2 -677.6352} C_DIS
LIN {X 20.2305,Y 24.0347,Z 62,A 43.4144,B 24.8137,C -3.1479,E1 25.101,E2 -680.6348} C_DIS
LIN {X 18.6195,Y 25.3035,Z 62,A 47.4217,B 24.8125,C -3.1577,E1 25.092,E2 -684.6507} C_DIS
LIN {X 16.1883,Y 26.9235,Z 62,A 52.2711,B 24.8122,C -3.1599,E1 25.0807,E2 -689.4898} C_DIS
LIN {X 14.9122,Y 27.6508,Z 62,A 55.4631,B 24.8111,C -3.1696,E1 25.0728,E2 -692.6956} C_DIS
LIN {X 12.2497,Y 28.9292,Z 62,A 60.1322,B 24.8114,C -3.1673,E1 25.061,E2 -697.3473} C_DIS
LIN {X 10.5532,Y 29.5906,Z 62,A 64.017,B 24.8102,C -3.1767,E1 25.0508,E2 -701.2464} C_DIS
LIN {X 8.5449,Y 30.2313,Z 62,A 67.4702,B 24.8104,C -3.175,E1 25.0416,E2 -704.6895} C_DIS
LIN {X 6.8794,Y 30.6538,Z 62,A 70.9039,B 24.8098,C -3.18,E1 25.0322,E2 -708.1302} C_DIS
LIN {X 4.404,Y 31.1055,Z 62,A 75.1084,B 24.8102,C -3.1773,E1 25.0207,E2 -712.3239} C_DIS
LIN {X 1.7103,Y 31.3691,Z 62,A 80.2025,B 24.8099,C -3.1793,E1 25.0065,E2 -717.4201} C_DIS
LIN {X -0.4128,Y 31.4134,Z 62,A 83.751,B 24.8104,C -3.1753,E1 24.9966,E2 -720.9587} C_DIS
LIN {X -2.0668,Y 31.3477,Z 62,A 86.8049,B 24.8104,C -3.1746,E1 24.9881,E2 -724.0117} C_DIS
LIN {X -3.8159,Y 31.1834,Z 62,A 90.3976,B 24.8102,C -3.1768,E1 24.9781,E2 -727.6118} C_DIS
LIN {X -5.4388,Y 30.9412,Z 62,A 93.4596,B 24.8104,C -3.1754,E1 24.9697,E2 -730.6733} C_DIS
LIN {X -7.5322,Y 30.4995,Z 62,A 96.9122,B 24.8113,C -3.1676,E1 24.9603,E2 -734.1119} C_DIS
LIN {X -9.2345,Y 30.0272,Z 62,A 100.292,B 24.8115,C -3.1657,E1 24.9512,E2 -737.4927} C_DIS
LIN {X -11.699,Y 29.1561,Z 62,A 106.1236,B 24.8111,C -3.1695,E1 24.936,E2 -743.3454} C_DIS
LIN {X -14.5234,Y 27.8574,Z 62,A 112.0711,B 24.8119,C -3.1631,E1 24.9211,E2 -749.2934} C_DIS
LIN {X -17.9817,Y 25.7606,Z 62,A 118.3488,B 24.8146,C -3.1398,E1 24.9065,E2 -755.5357} C_DIS
LIN {X -19.6083,Y 24.5448,Z 62,A 121.7905,B 24.8158,C -3.13,E1 24.8989,E2 -758.9664} C_DIS
LIN {X -20.6888,Y 23.6416,Z 62,A 124.3798,B 24.8164,C -3.1246,E1 24.8934,E2 -761.5528} C_DIS
LIN {X -21.6429,Y 22.7715,Z 62,A 127.2596,B 24.8166,C -3.1235,E1 24.8875,E2 -764.4419} C_DIS
LIN {X -23.2934,Y 21.0799,Z 62,A 131.7551,B 24.8176,C -3.1146,E1 24.8789,E2 -768.9357} C_DIS
LIN {X -25.1314,Y 18.8507,Z 62,A 136.5609,B 24.8196,C -3.0974,E1 24.8706,E2 -773.7229} C_DIS
LIN {X -26.1345,Y 17.4344,Z 62,A 140.6696,B 24.8198,C -3.0963,E1 24.8642,E2 -777.8494} C_DIS
LIN {X -28.1135,Y 14.0208,Z 62,A 146.8741,B 24.823,C -3.0682,E1 24.8559,E2 -784.0193} C_DIS
LIN {X -29.2654,Y 11.4215,Z 62,A 153.0061,B 24.824,C -3.0601,E1 24.8492,E2 -790.166} C_DIS
LIN {X -30.1082,Y 8.9691,Z 62,A 157.0277,B 24.8262,C -3.0404,E1 24.8458,E2 -794.1635} C_DIS
LIN {X -30.6096,Y 7.071,Z 62,A 161.1901,B 24.827,C -3.0337,E1 24.8431,E2 -798.3341} C_DIS
LIN {X -30.998,Y 5.1066,Z 62,A 164.4113,B 24.8287,C -3.0192,E1 24.8415,E2 -801.5396} C_DIS
LIN {X -31.241,Y 3.3088,Z 62,A 167.7689,B 24.8298,C -3.0092,E1 24.8404,E2 -804.8933} C_DIS
LIN {X -31.4041,Y 0.8607,Z 62,A 172.2942,B 24.8313,C -2.9956,E1 24.8398,E2 -809.4133} C_DIS
LIN {X -31.392,Y -1.2266,Z 62,A 175.9726,B 24.8328,C -2.9827,E1 24.84,E2 -813.0832} C_DIS
LIN {X -31.2557,Y -3.168,Z 62,A 179.5486,B 24.834,C -2.972,E1 24.8408,E2 -816.6548} C_DIS
LIN {X -31.0721,Y -4.6368,Z 62,A -177.9365,B 24.8351,C -2.9623,E1 24.8418,E2 -819.1616} C_DIS
LIN {X -30.8031,Y -6.1755,Z 62,A -174.7596,B 24.8358,C -2.9561,E1 24.8435,E2 -822.3426} C_DIS
LIN {X -30.3644,Y -8.0594,Z 62,A -170.6915,B 24.8365,C -2.9498,E1 24.8463,E2 -826.4192} C_DIS
LIN {X -29.3898,Y -11.099,Z 62,A -165.5634,B 24.8389,C -2.9276,E1 24.8509,E2 -831.5234} C_DIS
LIN {X -28.6774,Y -12.8281,Z 62,A -161.847,B 24.8397,C -2.9205,E1 24.855,E2 -835.2433} C_DIS
LIN {X -27.9224,Y -14.3979,Z 62,A -158.5667,B 24.8406,C -2.9128,E1 24.8591,E2 -838.5228} C_DIS
LIN {X -27.0373,Y -15.9978,Z 62,A -154.9831,B 24.8413,C -2.9061,E1 24.8641,E2 -842.1091} C_DIS
LIN {X -25.5641,Y -18.2599,Z 62,A -149.9129,B 24.8425,C -2.8953,E1 24.8721,E2 -847.1784} C_DIS
LIN {X -23.7124,Y -20.6076,Z 62,A -145.0085,B 24.8443,C -2.8783,E1 24.8808,E2 -852.0648} C_DIS
LIN {X -21.8045,Y -22.6162,Z 62,A -139.5786,B 24.8451,C -2.871,E1 24.8914,E2 -857.5007} C_DIS
LIN {X -19.7071,Y -24.4651,Z 62,A -134.0077,B 24.8457,C -2.8658,E1 24.9034,E2 -863.0805} C_DIS
LIN {X -17.9382,Y -25.7908,Z 62,A -129.8619,B 24.8463,C -2.8603,E1 24.9128,E2 -867.2274} C_DIS
LIN {X -14.9476,Y -27.6318,Z 62,A -124.3757,B 24.8482,C -2.8429,E1 24.926,E2 -872.6884} C_DIS
LIN {X -13.3369,Y -28.4441,Z 62,A -120.9796,B 24.8485,C -2.8401,E1 24.9345,E2 -876.0866} C_DIS
LIN {X -11.5349,Y -29.2214,Z 62,A -117.4715,B 24.8489,C -2.8358,E1 24.9436,E2 -879.5926} C_DIS
LIN {X -9.9108,Y -29.8118,Z 62,A -114.1313,B 24.8489,C -2.8352,E1 24.9524,E2 -882.9375} C_DIS
LIN {X -7.7491,Y -30.4451,Z 62,A -110.4967,B 24.8498,C -2.8279,E1 24.9621,E2 -886.5605} C_DIS
LIN {X -6.1015,Y -30.8179,Z 62,A -106.7546,B 24.8492,C -2.8333,E1 24.9724,E2 -890.3201} C_DIS
LIN {X -3.7941,Y -31.1861,Z 62,A -102.6361,B 24.8494,C -2.8309,E1 24.9838,E2 -894.4362} C_DIS
LIN {X -1.6274,Y -31.3735,Z 62,A -98.8808,B 24.8497,C -2.8287,E1 24.9942,E2 -898.1876} C_DIS
LIN {X 0.1406,Y -31.4146,Z 62,A -95.9275,B 24.8499,C -2.8264,E1 25.0025,E2 -901.1355} C_DIS
Enddeposition()
LIN {X 0.1406,Y -31.4146,Z 62,A -95.9275,B 24.8499,C -2.8264,E1 25.0025,E2 -901.1355} C_DIS
Startdeposition()
$VEL.CP = VEL_PRINT
LIN {X -1.173,Y -30.4137,Z 62,A -99.9206,B 24.8499,C -2.827,E1 24.9913,E2 -897.1435} C_DIS
LIN {X -3.3103,Y -30.2558,Z 62,A -103.9871,B 24.8499,C -2.827,E1 24.98,E2 -893.0748} C_DIS
LIN {X -5.3462,Y -29.9629,Z 62,A -108.3782,B 24.8503,C -2.8231,E1 24.9679,E2 -888.6702} C_DIS
LIN {X -8.5439,Y -29.2124,Z 62,A -114.1764,B 24.8495,C -2.8302,E1 24.9522,E2 -882.8805} C_DIS
LIN {X -10.2496,Y -28.6589,Z 62,A -116.9821,B 24.8487,C -2.8381,E1 24.9449,E2 -880.0884} C_DIS
LIN {X -12.1575,Y -27.9025,Z 62,A -121.7279,B 24.8491,C -2.834,E1 24.9326,E2 -875.322} C_DIS
LIN {X -14.2161,Y -26.912,Z 62,A -126.0376,B 24.8486,C -2.8392,E1 24.9219,E2 -871.0131} C_DIS
LIN {X -15.9424,Y -25.9272,Z 62,A -129.4023,B 24.8476,C -2.8477,E1 24.9138,E2 -867.6584} C_DIS
LIN {X -17.781,Y -24.7024,Z 62,A -133.9515,B 24.8473,C -2.8511,E1 24.9034,E2 -863.1018} C_DIS
LIN {X -19.9383,Y -22.9963,Z 62,A -138.2265,B 24.8455,C -2.8679,E1 24.8942,E2 -858.8506} C_DIS
LIN {X -21.3749,Y -21.6672,Z 62,A -142.9997,B 24.8456,C -2.8666,E1 24.8846,E2 -854.0546} C_DIS
LIN {X -23.7255,Y -19.0643,Z 62,A -149.3733,B 24.8438,C -2.8831,E1 24.873,E2 -847.6914} C_DIS
LIN {X -24.8715,Y -17.5434,Z 62,A -152.2503,B 24.8423,C -2.897,E1 24.8683,E2 -844.8337} C_DIS
LIN {X -25.748,Y -16.2299,Z 62,A -155.6143,B 24.8418,C -2.9015,E1 24.8632,E2 -841.4636} C_DIS
LIN {X -26.7549,Y -14.5096,Z 62,A -160.0866,B 24.8413,C -2.9061,E1 24.8571,E2 -836.9789} C_DIS
LIN {X -28.197,Y -11.4579,Z 62,A -165.2439,B 24.8384,C -2.9322,E1 24.8512,E2 -831.8557} C_DIS
LIN {X -28.7492,Y -9.9921,Z 62,A -169.0661,B 24.8382,C -2.9345,E1 24.8476,E2 -828.0174} C_DIS
LIN {X -29.5565,Y -7.2644,Z 62,A -174.1071,B 24.8362,C -2.9525,E1 24.8438,E2 -822.9901} C_DIS
LIN {X -30.0519,Y -4.8219,Z 62,A -179.2682,B 24.8349,C -2.9635,E1 24.8413,E2 -817.8249} C_DIS
LIN {X -30.3025,Y -2.8446,Z 62,A 177.6154,B 24.8332,C -2.9794,E1 24.8403,E2 -814.7278} C_DIS
LIN {X -30.4044,Y -1.3911,Z 62,A 174.5925,B 24.8324,C -2.986,E1 24.8398,E2 -811.7026} C_DIS
LIN {X -30.4288,Y 0.6761,Z 62,A 170.6746,B 24.8311,C -2.998,E1 24.8398,E2 -807.7897} C_DIS
LIN {X -30.2998,Y 2.8745,Z 62,A 166.7809,B 24.8294,C -3.0126,E1 24.8407,E2 -803.9078} C_DIS
LIN {X -30.0577,Y 4.7863,Z 62,A 163.2394,B 24.8281,C -3.0245,E1 24.842,E2 -800.3736} C_DIS
LIN {X -29.7389,Y 6.4767,Z 62,A 159.846,B 24.827,C -3.0335,E1 24.8439,E2 -796.9817} C_DIS
LIN {X -29.2575,Y 8.3882,Z 62,A 155.627,B 24.8261,C -3.0414,E1 24.8469,E2 -792.7571} C_DIS
LIN {X -28.6549,Y 10.2576,Z 62,A 152.0802,B 24.8247,C -3.0536,E1 24.8501,E2 -789.2193} C_DIS
LIN {X -27.8252,Y 12.3348,Z 62,A 147.7663,B 24.8234,C -3.0653,E1 24.8548,E2 -784.9095} C_DIS
LIN {X -26.4206,Y 15.11,Z 62,A 141.3569,B 24.8219,C -3.0782,E1 24.8632,E2 -778.4968} C_DIS
LIN {X -24.9182,Y 17.4772,Z 62,A 135.4989,B 24.8207,C -3.0883,E1 24.8724,E2 -772.634} C_DIS
LIN {X -22.1566,Y 20.8672,Z 62,A 128.3739,B 24.8173,C -3.1169,E1 24.8853,E2 -765.5451} C_DIS
LIN {X -20.6993,Y 22.3138,Z 62,A 124.5332,B 24.8163,C -3.126,E1 24.893,E2 -761.7102} C_DIS
LIN {X -19.2193,Y 23.6002,Z 62,A 120.632,B 24.8155,C -3.1323,E1 24.9014,E2 -757.8092} C_DIS
LIN {X -17.8033,Y 24.6864,Z 62,A 117.3411,B 24.8147,C -3.1396,E1 24.9088,E2 -754.5241} C_DIS
LIN {X -16.0462,Y 25.8624,Z 62,A 113.2726,B 24.8139,C -3.1463,E1 24.9183,E2 -750.4584} C_DIS
LIN {X -14.0488,Y 27.0001,Z 62,A 108.9533,B 24.813,C -3.1536,E1 24.9289,E2 -746.1442} C_DIS
LIN {X -11.1822,Y 28.3074,Z 62,A 102.5514,B 24.8125,C -3.158,E1 24.9453,E2 -739.7379} C_DIS
LIN {X -9.1195,Y 29.0373,Z 62,A 99.0685,B 24.8112,C -3.1683,E1 24.9545,E2 -736.2732} C_DIS
LIN {X -7.2077,Y 29.5703,Z 62,A 95.2196,B 24.8109,C -3.1709,E1 24.9649,E2 -732.4248} C_DIS
LIN {X -5.076,Y 30.0099,Z 62,A 90.8788,B 24.8109,C -3.1718,E1 24.9768,E2 -728.0816} C_DIS
LIN {X -2.3406,Y 30.3461,Z 62,A 86.1035,B 24.81,C -3.1784,E1 24.99,E2 -723.3191} C_DIS
LIN {X -0.3666,Y 30.4344,Z 62,A 82.1532,B 24.8102,C -3.1772,E1 25.0011,E2 -719.3655} C_DIS
LIN {X 1.7101,Y 30.388,Z 62,A 78.1881,B 24.8102,C -3.177,E1 25.0121,E2 -715.4009} C_DIS
LIN {X 3.6061,Y 30.2217,Z 62,A 74.6906,B 24.8102,C -3.1774,E1 25.0218,E2 -711.9066} C_DIS
LIN {X 5.6637,Y 29.9046,Z 62,A 70.7753,B 24.8103,C -3.1761,E1 25.0326,E2 -707.9924} C_DIS
LIN {X 7.7373,Y 29.4365,Z 62,A 67.0738,B 24.8102,C -3.1771,E1 25.0426,E2 -704.2985} C_DIS
LIN {X 9.0618,Y 29.0557,Z 62,A 64.5266,B 24.8103,C -3.1757,E1 25.0494,E2 -701.7526} C_DIS
LIN {X 10.5066,Y 28.5652,Z 62,A 61.4788,B 24.8109,C -3.1714,E1 25.0575,E2 -698.7006} C_DIS
LIN {X 12.827,Y 27.6011,Z 62,A 56.092,B 24.8123,C -3.1591,E1 25.0713,E2 -693.2977} C_DIS
LIN {X 14.6885,Y 26.6577,Z 62,A 52.5408,B 24.8124,C -3.1582,E1 25.08,E2 -689.7545} C_DIS
LIN {X 16.892,Y 25.3179,Z 62,A 47.6644,B 24.8133,C -3.1506,E1 25.0915,E2 -684.8759} C_DIS
LIN {X 18.9124,Y 23.8469,Z 62,A 42.7864,B 24.8146,C -3.1405,E1 25.1024,E2 -679.9915} C_DIS
LIN {X 20.654,Y 22.3557,Z 62,A 38.9139,B 24.8149,C -3.1374,E1 25.1104,E2 -676.1271} C_DIS
LIN {X 22.2311,Y 20.788,Z 62,A 34.4216,B 24.8164,C -3.1249,E1 25.1192,E2 -671.6245} C_DIS
LIN {X 23.5633,Y 19.2649,Z 62,A 30.7087,B 24.8173,C -3.1175,E1 25.1258,E2 -667.911} C_DIS
LIN {X 25.073,Y 17.2546,Z 62,A 26.3469,B 24.8181,C -3.1107,E1 25.133,E2 -663.5541} C_DIS
LIN {X 26.3738,Y 15.1913,Z 62,A 21.2038,B 24.8203,C -3.092,E1 25.1404,E2 -658.393} C_DIS
LIN {X 27.4837,Y 13.0771,Z 62,A 17.1289,B 24.8211,C -3.0851,E1 25.1455,E2 -654.3236} C_DIS
LIN {X 28.3104,Y 11.1748,Z 62,A 13.3592,B 24.8221,C -3.0759,E1 25.1495,E2 -650.5527} C_DIS
LIN {X 29.2065,Y 8.5639,Z 62,A 7.7108,B 24.8246,C -3.055,E1 25.1544,E2 -644.8868} C_DIS
LIN {X 29.8302,Y 6.0433,Z 62,A 3.8349,B 24.8247,C -3.0535,E1 25.1568,E2 -641.0299} C_DIS
LIN {X 30.0737,Y 4.6824,Z 62,A 1.1141,B 24.8258,C -3.044,E1 25.1581,E2 -638.3026} C_DIS
LIN {X 30.2768,Y 3.11,Z 62,A -2.2441,B 24.8274,C -3.0299,E1 25.1592,E2 -634.9308} C_DIS
LIN {X 30.4315,Y 0.5203,Z 62,A -7.3083,B 24.8294,C -3.0124,E1 25.1598,E2 -629.8551} C_DIS
LIN {X 30.3996,Y -1.477,Z 62,A -10.8703,B 24.8305,C -3.0032,E1 25.1594,E2 -626.2927} C_DIS
LIN {X 30.2618,Y -3.253,Z 62,A -14.1394,B 24.8315,C -2.9938,E1 25.1586,E2 -623.0207} C_DIS
LIN {X 29.9962,Y -5.1579,Z 62,A -17.8287,B 24.8329,C -2.9816,E1 25.157,E2 -619.3241} C_DIS
LIN {X 29.5941,Y -7.1102,Z 62,A -21.5289,B 24.8342,C -2.9706,E1 25.1547,E2 -615.6195} C_DIS
LIN {X 29.0334,Y -9.1341,Z 62,A -26.4556,B 24.8369,C -2.9459,E1 25.1507,E2 -610.6623} C_DIS
LIN {X 27.4997,Y -13.0438,Z 62,A -33.5793,B 24.8384,C -2.9326,E1 25.1429,E2 -603.5462} C_DIS
LIN {X 26.5073,Y -14.9569,Z 62,A -37.5934,B 24.8396,C -2.9216,E1 25.1376,E2 -599.5271} C_DIS
LIN {X 25.2609,Y -16.978,Z 62,A -41.8399,B 24.8406,C -2.9122,E1 25.1311,E2 -595.2795} C_DIS
LIN {X 24.0003,Y -18.7182,Z 62,A -45.9111,B 24.8418,C -2.9012,E1 25.1243,E2 -591.2018} C_DIS
LIN {X 22.6188,Y -20.3655,Z 62,A -50.0164,B 24.843,C -2.8903,E1 25.1167,E2 -587.0893} C_DIS
LIN {X 21.2576,Y -21.7827,Z 62,A -53.2908,B 24.8434,C -2.8868,E1 25.1103,E2 -583.8204} C_DIS
LIN {X 19.9927,Y -22.9488,Z 62,A -56.232,B 24.8438,C -2.8832,E1 25.1042,E2 -580.8824} C_DIS
LIN {X 18.7029,Y -24.0121,Z 62,A -59.8765,B 24.8452,C -2.8704,E1 25.0963,E2 -577.2212} C_DIS
LIN {X 17.1047,Y -25.1751,Z 62,A -63.6473,B 24.8461,C -2.8624,E1 25.0876,E2 -573.4445} C_DIS
LIN {X 15.4641,Y -26.2148,Z 62,A -67.0887,B 24.8465,C -2.8583,E1 25.0794,E2 -570.0042} C_DIS
LIN {X 13.7134,Y -27.172,Z 62,A -70.7084,B 24.847,C -2.8536,E1 25.0705,E2 -566.3837} C_DIS
LIN {X 12.2871,Y -27.8455,Z 62,A -73.8197,B 24.8477,C -2.8475,E1 25.0626,E2 -563.2656} C_DIS
LIN {X 10.0805,Y -28.7183,Z 62,A -78.8034,B 24.8489,C -2.8359,E1 25.0495,E2 -558.2649} C_DIS
LIN {X 8.4334,Y -29.2446,Z 62,A -81.6341,B 24.8488,C -2.837,E1 25.0419,E2 -555.4417} C_DIS
LIN {X 6.4532,Y -29.7441,Z 62,A -85.4438,B 24.8491,C -2.8338,E1 25.0316,E2 -551.6297} C_DIS
LIN {X 4.3578,Y -30.1226,Z 62,A -89.3442,B 24.8493,C -2.832,E1 25.0208,E2 -547.729} C_DIS
LIN {X 2.201,Y -30.3561,Z 62,A -93.2966,B 24.8494,C -2.8313,E1 25.0098,E2 -543.7772} C_DIS
LIN {X 0.3614,Y -30.4335,Z 62,A -97.432,B 24.8503,C -2.8233,E1 24.9982,E2 -539.6237} C_DIS
LIN {X 0.3614,Y -30.4335,Z 62,A -97.432,B 24.8503,C -2.8233,E1 24.9982,E2 -539.6237} C_DIS
Enddeposition()
LIN {X 0.1563,Y -29.456,Z 62,A -95.9616,B 24.8464,C -2.8592,E1 25.0026,E2 -541.1793} C_DIS
Startdeposition()
$VEL.CP = VEL_PRINT
LIN {X 2.0925,Y -29.3822,Z 62,A -91.5581,B 24.8455,C -2.8672,E1 25.0149,E2 -545.6005} C_DIS
LIN {X 4.1452,Y -29.1633,Z 62,A -87.893,B 24.8457,C -2.866,E1 25.0251,E2 -549.2597} C_DIS
LIN {X 5.8532,Y -28.8691,Z 62,A -84.4773,B 24.8453,C -2.8691,E1 25.0344,E2 -552.679} C_DIS
LIN {X 7.6952,Y -28.4335,Z 62,A -80.681,B 24.8448,C -2.8741,E1 25.0447,E2 -556.4813} C_DIS
LIN {X 9.0419,Y -28.0344,Z 62,A -77.6841,B 24.8441,C -2.8802,E1 25.0527,E2 -559.4873} C_DIS
LIN {X 11.2395,Y -27.2282,Z 62,A -73.5213,B 24.844,C -2.8819,E1 25.0635,E2 -563.6449} C_DIS
LIN {X 13.0722,Y -26.3969,Z 62,A -69.5423,B 24.8432,C -2.8887,E1 25.0736,E2 -567.6297} C_DIS
LIN {X 14.6904,Y -25.5318,Z 62,A -66.0343,B 24.8426,C -2.8941,E1 25.0822,E2 -571.1403} C_DIS
LIN {X 16.4634,Y -24.4262,Z 62,A -62.0297,B 24.8419,C -2.901,E1 25.0916,E2 -575.1483} C_DIS
LIN {X 17.9966,Y -23.3196,Z 62,A -58.2457,B 24.8409,C -2.9099,E1 25.1,E2 -578.9396} C_DIS
LIN {X 19.5702,Y -22.0159,Z 62,A -54.6436,B 24.8404,C -2.914,E1 25.1077,E2 -582.5377} C_DIS
LIN {X 20.7028,Y -20.9541,Z 62,A -51.1581,B 24.839,C -2.9269,E1 25.1147,E2 -586.039} C_DIS
LIN {X 22.1765,Y -19.3877,Z 62,A -47.1455,B 24.8381,C -2.935,E1 25.1222,E2 -590.0532} C_DIS
LIN {X 23.3846,Y -17.9122,Z 62,A -43.6375,B 24.8373,C -2.9421,E1 25.1283,E2 -593.5615} C_DIS
LIN {X 24.5181,Y -16.3267,Z 62,A -39.7465,B 24.8361,C -2.9536,E1 25.1345,E2 -597.4606} C_DIS
LIN {X 25.4609,Y -14.8137,Z 62,A -36.6352,B 24.8355,C -2.9587,E1 25.139,E2 -600.5682} C_DIS
LIN {X 26.2006,Y -13.4616,Z 62,A -33.5597,B 24.8344,C -2.9683,E1 25.1431,E2 -603.6502} C_DIS
LIN {X 26.9951,Y -11.7875,Z 62,A -29.3834,B 24.8324,C -2.9863,E1 25.1479,E2 -607.8465} C_DIS
LIN {X 27.8514,Y -9.5922,Z 62,A -25.0198,B 24.8312,C -2.9972,E1 25.1521,E2 -612.2115} C_DIS
LIN {X 28.443,Y -7.6601,Z 62,A -21.4301,B 24.8303,C -3.0048,E1 25.1549,E2 -615.7986} C_DIS
LIN {X 28.8701,Y -5.8483,Z 62,A -17.5692,B 24.8287,C -3.0192,E1 25.1572,E2 -619.6711} C_DIS
LIN {X 29.1936,Y -3.9286,Z 62,A -13.828,B 24.8274,C -3.0304,E1 25.1587,E2 -623.4168} C_DIS
LIN {X 29.404,Y -1.7613,Z 62,A -10.1596,B 24.8267,C -3.0362,E1 25.1596,E2 -627.0774} C_DIS
LIN {X 29.4546,Y -0.3594,Z 62,A -6.4048,B 24.8242,C -3.0582,E1 25.1598,E2 -630.8619} C_DIS
LIN {X 29.3743,Y 2.203,Z 62,A -2.0622,B 24.8234,C -3.0653,E1 25.1591,E2 -635.1954} C_DIS
LIN {X 29.172,Y 4.0839,Z 62,A 1.5489,B 24.8222,C -3.0757,E1 25.1579,E2 -638.8098} C_DIS
LIN {X 28.8376,Y 6.0064,Z 62,A 4.6605,B 24.8219,C -3.0783,E1 25.1563,E2 -641.9095} C_DIS
LIN {X 28.275,Y 8.2594,Z 62,A 9.3929,B 24.82,C -3.0945,E1 25.153,E2 -646.6529} C_DIS
LIN {X 27.8097,Y 9.711,Z 62,A 12.7449,B 24.8184,C -3.1081,E1 25.1501,E2 -650.0182} C_DIS
LIN {X 27.1537,Y 11.4174,Z 62,A 16.2736,B 24.8172,C -3.1178,E1 25.1464,E2 -653.5503} C_DIS
LIN {X 26.3398,Y 13.1874,Z 62,A 20.289,B 24.8157,C -3.131,E1 25.1415,E2 -657.5754} C_DIS
LIN {X 25.0804,Y 15.4494,Z 62,A 25.2268,B 24.8143,C -3.1428,E1 25.1346,E2 -662.5158} C_DIS
LIN {X 23.8605,Y 17.2738,Z 62,A 29.0535,B 24.8137,C -3.1478,E1 25.1285,E2 -666.3355} C_DIS
LIN {X 22.8367,Y 18.6056,Z 62,A 32.3301,B 24.8128,C -3.1555,E1 25.1228,E2 -669.6151} C_DIS
LIN {X 21.2888,Y 20.3588,Z 62,A 37.7758,B 24.8103,C -3.1762,E1 25.1125,E2 -675.0859} C_DIS
LIN {X 19.7914,Y 21.8177,Z 62,A 41.3072,B 24.8101,C -3.1779,E1 25.1053,E2 -678.6068} C_DIS
LIN {X 18.2376,Y 23.1312,Z 62,A 44.6645,B 24.8101,C -3.1781,E1 25.0981,E2 -681.9519} C_DIS
LIN {X 16.8485,Y 24.1622,Z 62,A 48.6871,B 24.8085,C -3.1913,E1 25.0889,E2 -685.9916} C_DIS
LIN {X 14.6623,Y 25.5479,Z 62,A 53.5304,B 24.8079,C -3.1964,E1 25.0774,E2 -690.832} C_DIS
LIN {X 12.8438,Y 26.509,Z 62,A 57.5714,B 24.8072,C -3.2018,E1 25.0673,E2 -694.8747} C_DIS
LIN {X 11.3687,Y 27.1742,Z 62,A 60.3843,B 24.8072,C -3.2015,E1 25.0601,E2 -697.6801} C_DIS
LIN {X 9.91,Y 27.7397,Z 62,A 63.5345,B 24.8068,C -3.2054,E1 25.0519,E2 -700.8329} C_DIS
LIN {X 8.2917,Y 28.2655,Z 62,A 66.8587,B 24.8065,C -3.208,E1 25.043,E2 -704.1573} C_DIS
LIN {X 6.4968,Y 28.7313,Z 62,A 70.4977,B 24.8062,C -3.2103,E1 25.0331,E2 -707.7965} C_DIS
LIN {X 4.258,Y 29.1473,Z 62,A 75.4218,B 24.8054,C -3.2167,E1 25.0195,E2 -712.731} C_DIS
LIN {X 1.7099,Y 29.4069,Z 62,A 80.0772,B 24.8058,C -3.2138,E1 25.0066,E2 -717.377} C_DIS
LIN {X -0.213,Y 29.4557,Z 62,A 83.5974,B 24.8061,C -3.211,E1 24.9968,E2 -720.8902} C_DIS
LIN {X -2.1693,Y 29.3769,Z 62,A 87.6355,B 24.806,C -3.2118,E1 24.9855,E2 -724.9313} C_DIS
LIN {X -3.8544,Y 29.2032,Z 62,A 91.329,B 24.8058,C -3.2136,E1 24.9753,E2 -728.6317} C_DIS
LIN {X -6.3456,Y 28.7649,Z 62,A 95.7382,B 24.8068,C -3.205,E1 24.9633,E2 -733.0256} C_DIS
LIN {X -8.1101,Y 28.3181,Z 62,A 98.9755,B 24.8076,C -3.1989,E1 24.9546,E2 -736.253} C_DIS
LIN {X -9.3177,Y 27.9441,Z 62,A 101.7137,B 24.8076,C -3.1985,E1 24.9473,E2 -738.9952} C_DIS
LIN {X -11.2295,Y 27.2323,Z 62,A 105.8253,B 24.8081,C -3.1945,E1 24.9366,E2 -743.1061} C_DIS
LIN {X -13.106,Y 26.3802,Z 62,A 109.7057,B 24.8089,C -3.1873,E1 24.9268,E2 -746.9793} C_DIS
LIN {X -14.8339,Y 25.4493,Z 62,A 113.7492,B 24.8095,C -3.1827,E1 24.917,E2 -751.0235} C_DIS
LIN {X -16.6935,Y 24.2699,Z 62,A 117.3504,B 24.8111,C -3.1693,E1 24.9086,E2 -754.6044} C_DIS
LIN {X -17.7968,Y 23.4718,Z 62,A 120.3426,B 24.8114,C -3.1667,E1 24.9018,E2 -757.6008} C_DIS
LIN {X -18.9845,Y 22.5232,Z 62,A 123.3954,B 24.8121,C -3.1611,E1 24.8953,E2 -760.6519} C_DIS
LIN {X -20.2032,Y 21.4362,Z 62,A 127.1219,B 24.8125,C -3.1581,E1 24.8876,E2 -764.3864} C_DIS
LIN {X -21.7263,Y 19.8909,Z 62,A 131.9815,B 24.8131,C -3.1527,E1 24.8784,E2 -769.2544} C_DIS
LIN {X -24.025,Y 17.0437,Z 62,A 138.0981,B 24.8162,C -3.1269,E1 24.868,E2 -775.3383} C_DIS
LIN {X -25.0368,Y 15.5186,Z 62,A 141.9146,B 24.8171,C -3.119,E1 24.8623,E2 -779.1552} C_DIS
LIN {X -26.2965,Y 13.2739,Z 62,A 146.7795,B 24.8189,C -3.1037,E1 24.8559,E2 -784.0093} C_DIS
LIN {X -27.0852,Y 11.5802,Z 62,A 150.5977,B 24.82,C -3.0944,E1 24.8515,E2 -787.826} C_DIS
LIN {X -27.8654,Y 9.551,Z 62,A 154.7474,B 24.8215,C -3.0811,E1 24.8476,E2 -791.9676} C_DIS
LIN {X -28.5202,Y 7.3676,Z 62,A 159.3952,B 24.8229,C -3.069,E1 24.8441,E2 -796.6133} C_DIS
LIN {X -29.0122,Y 5.0976,Z 62,A 163.4398,B 24.8249,C -3.0518,E1 24.8419,E2 -800.6406} C_DIS
LIN {X -29.2024,Y 3.8604,Z 62,A 166.3199,B 24.8254,C -3.0472,E1 24.8408,E2 -803.5269} C_DIS
LIN {X -29.4053,Y 1.7383,Z 62,A 170.3568,B 24.827,C -3.0335,E1 24.8399,E2 -807.5552} C_DIS
LIN {X -29.455,Y -0.3474,Z 62,A 174.6251,B 24.8283,C -3.0223,E1 24.8399,E2 -811.8223} C_DIS
LIN {X -29.3274,Y -2.7542,Z 62,A 179.5256,B 24.8298,C -3.0092,E1 24.8409,E2 -816.7209} C_DIS
LIN {X -28.9129,Y -5.6327,Z 62,A -175.1458,B 24.832,C -2.9897,E1 24.8433,E2 -822.0345} C_DIS
LIN {X -28.4701,Y -7.5598,Z 62,A -171.3944,B 24.8334,C -2.9776,E1 24.8458,E2 -825.7789} C_DIS
LIN {X -27.9145,Y -9.4046,Z 62,A -167.6131,B 24.8346,C -2.967,E1 24.849,E2 -829.5563} C_DIS
LIN {X -27.2623,Y -11.1556,Z 62,A -163.7477,B 24.8355,C -2.9583,E1 24.8529,E2 -833.4226} C_DIS
LIN {X -26.5374,Y -12.7846,Z 62,A -160.1563,B 24.8365,C -2.9497,E1 24.8571,E2 -837.013} C_DIS
LIN {X -25.5261,Y -14.7003,Z 62,A -156.0516,B 24.8378,C -2.9378,E1 24.8627,E2 -841.111} C_DIS
LIN {X -24.4643,Y -16.4072,Z 62,A -152.3014,B 24.839,C -2.9269,E1 24.8683,E2 -844.8539} C_DIS
LIN {X -23.4698,Y -17.8005,Z 62,A -149.0542,B 24.84,C -2.9183,E1 24.8737,E2 -848.0963} C_DIS
LIN {X -22.2862,Y -19.2621,Z 62,A -145.0022,B 24.8405,C -2.9131,E1 24.8809,E2 -852.1543} C_DIS
LIN {X -20.836,Y -20.8224,Z 62,A -140.9132,B 24.8415,C -2.9039,E1 24.8889,E2 -856.2392} C_DIS
LIN {X -19.3801,Y -22.1831,Z 62,A -137.2012,B 24.8425,C -2.8951,E1 24.8965,E2 -859.9451} C_DIS
LIN {X -18.2922,Y -23.0883,Z 62,A -134.2909,B 24.8429,C -2.8915,E1 24.9029,E2 -862.8576} C_DIS
LIN {X -16.6154,Y -24.3233,Z 62,A -130.2043,B 24.8436,C -2.8852,E1 24.9122,E2 -866.9433} C_DIS
LIN {X -14.8256,Y -25.4541,Z 62,A -125.9861,B 24.8441,C -2.8802,E1 24.9222,E2 -871.1625} C_DIS
LIN {X -13.1196,Y -26.3734,Z 62,A -122.7881,B 24.8452,C -2.8705,E1 24.9301,E2 -874.3463} C_DIS
LIN {X -11.3219,Y -27.1939,Z 62,A -118.033,B 24.8447,C -2.8747,E1 24.9423,E2 -879.1224} C_DIS
LIN {X -9.5252,Y -27.8741,Z 62,A -115.0088,B 24.8458,C -2.865,E1 24.9502,E2 -882.1296} C_DIS
LIN {X -8.3558,Y -28.2463,Z 62,A -112.453,B 24.8458,C -2.865,E1 24.9571,E2 -884.6896} C_DIS
LIN {X -6.6152,Y -28.704,Z 62,A -108.7527,B 24.8458,C -2.865,E1 24.9671,E2 -888.3951} C_DIS
LIN {X -4.5659,Y -29.1005,Z 62,A -104.8887,B 24.8461,C -2.8618,E1 24.9777,E2 -892.2554} C_DIS
LIN {X -2.9449,Y -29.3091,Z 62,A -101.4969,B 24.8459,C -2.8635,E1 24.9872,E2 -895.6534} C_DIS
LIN {X -0.8805,Y -29.4433,Z 62,A -97.4934,B 24.8459,C -2.8635,E1 24.9983,E2 -899.6582} C_DIS
LIN {X -0.8805,Y -29.4433,Z 62,A -97.4934,B 24.8459,C -2.8635,E1 24.9983,E2 -899.6582} C_DIS
Enddeposition()
LIN {X 0.162,Y -28.4735,Z 62,A -97.1224,B 24.8459,C -2.8645,E1 24.9994,E2 -900.0312} C_DIS
Startdeposition()
$VEL.CP = VEL_PRINT
LIN {X -1.7168,Y -28.4253,Z 62,A -101.3172,B 24.8463,C -2.8601,E1 24.9877,E2 -895.8253} C_DIS
LIN {X -3.8332,Y -28.2181,Z 62,A -105.5707,B 24.8463,C -2.8609,E1 24.9759,E2 -891.5709} C_DIS
LIN {X -5.8931,Y -27.8608,Z 62,A -109.8086,B 24.8461,C -2.8622,E1 24.9642,E2 -887.3314} C_DIS
LIN {X -7.984,Y -27.3349,Z 62,A -114.0499,B 24.8457,C -2.8656,E1 24.9528,E2 -883.0918} C_DIS
LIN {X -9.9249,Y -26.6918,Z 62,A -118.243,B 24.8454,C -2.8683,E1 24.9418,E2 -878.8969} C_DIS
LIN {X -11.878,Y -25.8817,Z 62,A -122.4759,B 24.8449,C -2.873,E1 24.9309,E2 -874.6651} C_DIS
LIN {X -13.7103,Y -24.9595,Z 62,A -126.6542,B 24.8444,C -2.8777,E1 24.9206,E2 -870.4866} C_DIS
LIN {X -15.5324,Y -23.8684,Z 62,A -130.9411,B 24.8437,C -2.8839,E1 24.9104,E2 -866.2008} C_DIS
LIN {X -17.2401,Y -22.6657,Z 62,A -135.2005,B 24.843,C -2.8904,E1 24.9008,E2 -861.9421} C_DIS
LIN {X -18.8642,Y -21.333,Z 62,A -139.4264,B 24.8422,C -2.8983,E1 24.8919,E2 -857.7186} C_DIS
LIN {X -20.3737,Y -19.8964,Z 62,A -143.6341,B 24.8412,C -2.9067,E1 24.8835,E2 -853.5133} C_DIS
LIN {X -21.7751,Y -18.3519,Z 62,A -147.7326,B 24.8402,C -2.9166,E1 24.876,E2 -849.4201} C_DIS
LIN {X -23.0648,Y -16.7022,Z 62,A -152.1081,B 24.8392,C -2.9255,E1 24.8686,E2 -845.0448} C_DIS
LIN {X -24.2258,Y -14.9685,Z 62,A -156.3047,B 24.838,C -2.936,E1 24.8623,E2 -840.8521} C_DIS
LIN {X -25.2763,Y -13.1174,Z 62,A -160.6606,B 24.8368,C -2.9468,E1 24.8565,E2 -836.4991} C_DIS
LIN {X -26.1911,Y -11.1789,Z 62,A -164.8975,B 24.8354,C -2.9592,E1 24.8516,E2 -832.2686} C_DIS
LIN {X -26.9238,Y -9.2769,Z 62,A -169.0795,B 24.8342,C -2.9704,E1 24.8476,E2 -828.0898} C_DIS
LIN {X -27.5289,Y -7.2875,Z 62,A -173.3,B 24.8328,C -2.9825,E1 24.8444,E2 -823.8738} C_DIS
LIN {X -27.9944,Y -5.2219,Z 62,A -177.585,B 24.8314,C -2.9952,E1 24.842,E2 -819.5939} C_DIS
LIN {X -28.3006,Y -3.1662,Z 62,A 178.206,B 24.83,C -3.0078,E1 24.8405,E2 -815.39} C_DIS
LIN {X -28.4579,Y -1.0495,Z 62,A 173.8837,B 24.8285,C -3.0207,E1 24.8398,E2 -811.0727} C_DIS
LIN {X -28.4593,Y 1.0065,Z 62,A 169.7021,B 24.827,C -3.0334,E1 24.84,E2 -806.8962} C_DIS
LIN {X -28.3086,Y 3.0926,Z 62,A 165.4818,B 24.8255,C -3.0465,E1 24.8411,E2 -802.6819} C_DIS
LIN {X -27.9962,Y 5.2125,Z 62,A 161.1054,B 24.824,C -3.0595,E1 24.8431,E2 -798.3106} C_DIS
LIN {X -27.5402,Y 7.2449,Z 62,A 156.9247,B 24.8225,C -3.0724,E1 24.8458,E2 -794.1366} C_DIS
LIN {X -26.9242,Y 9.2758,Z 62,A 152.6248,B 24.8211,C -3.0852,E1 24.8495,E2 -789.8426} C_DIS
LIN {X -26.1721,Y 11.2239,Z 62,A 148.3929,B 24.8196,C -3.0975,E1 24.854,E2 -785.6165} C_DIS
LIN {X -25.2953,Y 13.0802,Z 62,A 144.4002,B 24.8181,C -3.1102,E1 24.8589,E2 -781.6329} C_DIS
LIN {X -24.5177,Y 14.4847,Z 62,A 141.1006,B 24.8171,C -3.1189,E1 24.8635,E2 -778.3366} C_DIS
LIN {X -23.4692,Y 16.129,Z 62,A 137.0064,B 24.816,C -3.1284,E1 24.8698,E2 -774.2448} C_DIS
LIN {X -22.2283,Y 17.8004,Z 62,A 132.8247,B 24.8147,C -3.1393,E1 24.8769,E2 -770.0693} C_DIS
LIN {X -20.8603,Y 19.3856,Z 62,A 128.5838,B 24.8135,C -3.1494,E1 24.8848,E2 -765.8337} C_DIS
LIN {X -19.3543,Y 20.8892,Z 62,A 124.2874,B 24.8123,C -3.1592,E1 24.8934,E2 -761.5429} C_DIS
LIN {X -17.7712,Y 22.2516,Z 62,A 120.0547,B 24.8113,C -3.168,E1 24.9025,E2 -757.3151} C_DIS
LIN {X -16.1262,Y 23.4711,Z 62,A 115.9082,B 24.8103,C -3.1759,E1 24.9119,E2 -753.1731} C_DIS
LIN {X -14.3337,Y 24.6069,Z 62,A 111.6218,B 24.8094,C -3.1834,E1 24.9221,E2 -748.8914} C_DIS
LIN {X -12.4925,Y 25.5909,Z 62,A 107.4268,B 24.8086,C -3.1901,E1 24.9325,E2 -744.7011} C_DIS
LIN {X -10.5844,Y 26.4372,Z 62,A 103.1882,B 24.8079,C -3.1957,E1 24.9434,E2 -740.466} C_DIS
LIN {X -8.5954,Y 27.1491,Z 62,A 98.9236,B 24.8074,C -3.2006,E1 24.9547,E2 -736.2051} C_DIS
LIN {X -6.5782,Y 27.7071,Z 62,A 94.7025,B 24.8069,C -3.2046,E1 24.9661,E2 -731.9873} C_DIS
LIN {X -4.5438,Y 28.1123,Z 62,A 90.5333,B 24.8065,C -3.2077,E1 24.9775,E2 -727.8214} C_DIS
LIN {X -2.47,Y 28.3698,Z 62,A 86.2806,B 24.8063,C -3.2095,E1 24.9893,E2 -723.5703} C_DIS
LIN {X -0.3811,Y 28.4746,Z 62,A 82.0785,B 24.8061,C -3.2107,E1 25.0011,E2 -719.3707} C_DIS
LIN {X 1.7456,Y 28.4237,Z 62,A 77.7209,B 24.8061,C -3.2103,E1 25.0132,E2 -715.0133} C_DIS
LIN {X 3.9359,Y 28.2035,Z 62,A 73.4531,B 24.8061,C -3.211,E1 25.025,E2 -710.7504} C_DIS
LIN {X 5.8759,Y 27.8644,Z 62,A 69.3715,B 24.8064,C -3.2083,E1 25.0362,E2 -706.6671} C_DIS
LIN {X 7.9421,Y 27.3473,Z 62,A 65.1621,B 24.8067,C -3.2064,E1 25.0476,E2 -702.4598} C_DIS
LIN {X 9.911,Y 26.6969,Z 62,A 60.9858,B 24.8071,C -3.2028,E1 25.0586,E2 -698.2834} C_DIS
LIN {X 11.8694,Y 25.8857,Z 62,A 56.7615,B 24.8076,C -3.1987,E1 25.0694,E2 -694.0594} C_DIS
LIN {X 13.7009,Y 24.9646,Z 62,A 52.6167,B 24.8082,C -3.1932,E1 25.0796,E2 -689.9133} C_DIS
LIN {X 15.4067,Y 23.9491,Z 62,A 48.765,B 24.8088,C -3.1888,E1 25.0888,E2 -686.0635} C_DIS
LIN {X 17.0119,Y 22.8371,Z 62,A 44.7718,B 24.8096,C -3.1816,E1 25.0978,E2 -682.0671} C_DIS
LIN {X 18.5982,Y 21.5653,Z 62,A 40.6425,B 24.8106,C -3.1736,E1 25.1067,E2 -677.9347} C_DIS
LIN {X 20.1638,Y 20.1088,Z 62,A 36.3826,B 24.8116,C -3.1654,E1 25.1153,E2 -673.6731} C_DIS
LIN {X 21.5694,Y 18.5933,Z 62,A 32.2113,B 24.8127,C -3.1562,E1 25.123,E2 -669.4983} C_DIS
LIN {X 22.8789,Y 16.9561,Z 62,A 28.0604,B 24.8138,C -3.147,E1 25.1301,E2 -665.3454} C_DIS
LIN {X 24.0373,Y 15.2692,Z 62,A 23.911,B 24.815,C -3.1364,E1 25.1365,E2 -661.1915} C_DIS
LIN {X 25.1051,Y 13.4418,Z 62,A 19.7045,B 24.8163,C -3.1258,E1 25.1423,E2 -656.9819} C_DIS
LIN {X 26.0194,Y 11.5731,Z 62,A 15.5139,B 24.8176,C -3.1143,E1 25.1472,E2 -652.7865} C_DIS
LIN {X 26.8114,Y 9.597,Z 62,A 11.2827,B 24.819,C -3.1027,E1 25.1514,E2 -648.5515} C_DIS
LIN {X 27.4506,Y 7.5771,Z 62,A 7.0543,B 24.8204,C -3.0907,E1 25.1548,E2 -644.3186} C_DIS
LIN {X 27.9321,Y 5.5455,Z 62,A 2.9077,B 24.8218,C -3.0787,E1 25.1572,E2 -640.1678} C_DIS
LIN {X 28.2588,Y 3.5191,Z 62,A -1.2244,B 24.8233,C -3.066,E1 25.1589,E2 -636.03} C_DIS
LIN {X 28.4427,Y 1.4023,Z 62,A -5.4449,B 24.8247,C -3.0534,E1 25.1597,E2 -631.8048} C_DIS
LIN {X 28.4684,Y -0.7094,Z 62,A -9.6593,B 24.8262,C -3.0406,E1 25.1597,E2 -627.585} C_DIS
LIN {X 28.3396,Y -2.7966,Z 62,A -13.8658,B 24.8277,C -3.0274,E1 25.1587,E2 -623.3723} C_DIS
LIN {X 28.058,Y -4.8686,Z 62,A -18.0209,B 24.8291,C -3.015,E1 25.1569,E2 -619.2121} C_DIS
LIN {X 27.6336,Y -6.8794,Z 62,A -22.151,B 24.8306,C -3.0022,E1 25.1543,E2 -615.0758} C_DIS
LIN {X 27.0545,Y -8.888,Z 62,A -26.3277,B 24.832,C -2.9898,E1 25.1509,E2 -610.8934} C_DIS
LIN {X 26.3301,Y -10.8473,Z 62,A -30.5282,B 24.8334,C -2.9772,E1 25.1466,E2 -606.6865} C_DIS
LIN {X 25.4602,Y -12.7561,Z 62,A -34.7183,B 24.8347,C -2.9653,E1 25.1416,E2 -602.4907} C_DIS
LIN {X 24.4402,Y -14.6158,Z 62,A -38.9656,B 24.8361,C -2.9535,E1 25.1357,E2 -598.2374} C_DIS
LIN {X 23.2806,Y -16.4003,Z 62,A -43.1668,B 24.8373,C -2.9429,E1 25.1291,E2 -594.0318} C_DIS
LIN {X 22.0138,Y -18.0651,Z 62,A -47.3659,B 24.8384,C -2.9321,E1 25.1218,E2 -589.8268} C_DIS
LIN {X 20.6283,Y -19.6323,Z 62,A -51.5634,B 24.8396,C -2.9219,E1 25.1139,E2 -585.6237} C_DIS
LIN {X 19.1188,Y -21.1051,Z 62,A -55.7688,B 24.8406,C -2.9125,E1 25.1053,E2 -581.4133} C_DIS
LIN {X 17.5177,Y -22.4518,Z 62,A -59.9484,B 24.8416,C -2.9039,E1 25.0963,E2 -577.2291} C_DIS
LIN {X 15.8221,Y -23.6773,Z 62,A -64.1548,B 24.8425,C -2.8956,E1 25.0866,E2 -573.0175} C_DIS
LIN {X 14.2272,Y -24.6681,Z 62,A -67.8666,B 24.8431,C -2.8896,E1 25.0777,E2 -569.3028} C_DIS
LIN {X 12.4568,Y -25.6081,Z 62,A -71.8855,B 24.8438,C -2.8832,E1 25.0677,E2 -565.2797} C_DIS
LIN {X 10.5822,Y -26.4381,Z 62,A -76.0862,B 24.8445,C -2.8765,E1 25.0569,E2 -561.0731} C_DIS
LIN {X 8.5887,Y -27.1512,Z 62,A -80.3056,B 24.8451,C -2.8717,E1 25.0457,E2 -556.8506} C_DIS
LIN {X 6.5734,Y -27.7082,Z 62,A -84.5049,B 24.8455,C -2.8676,E1 25.0344,E2 -552.6479} C_DIS
LIN {X 4.5568,Y -28.1102,Z 62,A -88.636,B 24.8458,C -2.8645,E1 25.023,E2 -548.5138} C_DIS
LIN {X 2.4581,Y -28.3709,Z 62,A -92.9189,B 24.8461,C -2.8618,E1 25.0111,E2 -544.2275} C_DIS
LIN {X 0.3731,Y -28.4747,Z 62,A -97.1131,B 24.8463,C -2.8605,E1 24.9994,E2 -540.0312} C_DIS
LIN {X 0.3731,Y -28.4747,Z 62,A -97.1131,B 24.8463,C -2.8605,E1 24.9994,E2 -540.0312} C_DIS
Enddeposition()
LIN {X 0.1498,Y -30.5866,Z 66.5315,A -97.1089,B 24.8465,C -2.8588,E1 24.9994,E2 -540.0312} C_DIS
LIN {X 0.1131,Y -36.9257,Z 80.1262,A -97.073,B 24.8481,C -2.8437,E1 24.9994,E2 -540.0312} C_DIS
LIN {X 0.1131,Y -36.9257,Z 101.1262,A -97.4223,B 24.8319,C -2.9904,E1 24.9994,E2 -540.0312} C_DIS
LIN {X 0.2575,Y -56.3798,Z 101.1262,A -96.1097,B 24.8661,C -2.6701,E1 25.0009,E2 -540.5817} C_DIS
LIN {X 0.2575,Y -56.3798,Z 81.1262,A -95.7774,B 24.8798,C -2.5304,E1 25.0009,E2 -540.5817} C_DIS
LIN {X 0.2333,Y -50.0406,Z 67.5315,A -95.8101,B 24.8785,C -2.5441,E1 25.0009,E2 -540.5817} C_DIS
LIN {X 0.2252,Y -47.9275,Z 63,A -95.8225,B 24.878,C -2.5494,E1 25.0009,E2 -540.5817} C_DIS
Startdeposition()
$VEL.CP = VEL_PRINT
LIN {X -1.7211,Y -47.9012,Z 63,A -98.7904,B 24.8791,C -2.5383,E1 24.9926,E2 -537.5872} C_DIS
LIN {X -4.1125,Y -47.7556,Z 63,A -101.6409,B 24.8791,C -2.5385,E1 24.9846,E2 -534.7361} C_DIS
LIN {X -6.4508,Y -47.4963,Z 63,A -104.4543,B 24.879,C -2.539,E1 24.9768,E2 -531.9218} C_DIS
LIN {X -8.7735,Y -47.1226,Z 63,A -107.2688,B 24.879,C -2.5398,E1 24.9691,E2 -529.1065} C_DIS
LIN {X -11.0752,Y -46.6353,Z 63,A -110.0843,B 24.8788,C -2.541,E1 24.9614,E2 -526.2904} C_DIS
LIN {X -13.3501,Y -46.0357,Z 63,A -112.9008,B 24.8786,C -2.5427,E1 24.9538,E2 -523.4735} C_DIS
LIN {X -15.5929,Y -45.3252,Z 63,A -115.7182,B 24.8784,C -2.5448,E1 24.9464,E2 -520.6559} C_DIS
LIN {X -17.7981,Y -44.5055,Z 63,A -118.5366,B 24.8782,C -2.5473,E1 24.939,E2 -517.8374} C_DIS
LIN {X -19.9605,Y -43.5786,Z 63,A -121.3561,B 24.8779,C -2.5502,E1 24.9318,E2 -515.018} C_DIS
LIN {X -22.0747,Y -42.5467,Z 63,A -124.1762,B 24.8776,C -2.5535,E1 24.9248,E2 -512.1982} C_DIS
LIN {X -23.9794,Y -41.5021,Z 63,A -126.7887,B 24.8773,C -2.5567,E1 24.9184,E2 -509.5858} C_DIS
LIN {X -26.1387,Y -40.1781,Z 63,A -129.8196,B 24.8769,C -2.5612,E1 24.9113,E2 -506.556} C_DIS
LIN {X -28.0787,Y -38.8472,Z 63,A -132.6426,B 24.8764,C -2.5656,E1 24.9048,E2 -503.7338} C_DIS
LIN {X -29.9279,Y -37.4409,Z 63,A -135.4401,B 24.876,C -2.5701,E1 24.8987,E2 -500.9368} C_DIS
LIN {X -31.7512,Y -35.9079,Z 63,A -138.291,B 24.8755,C -2.5754,E1 24.8926,E2 -498.0875} C_DIS
LIN {X -33.4748,Y -34.3067,Z 63,A -141.1165,B 24.8749,C -2.5809,E1 24.8869,E2 -495.2634} C_DIS
LIN {X -35.0972,Y -32.6448,Z 63,A -143.9159,B 24.8744,C -2.5865,E1 24.8815,E2 -492.465} C_DIS
LIN {X -36.6763,Y -30.8604,Z 63,A -146.7695,B 24.8738,C -2.5927,E1 24.8763,E2 -489.6135} C_DIS
LIN {X -38.1464,Y -29.0236,Z 63,A -149.5972,B 24.8732,C -2.5991,E1 24.8715,E2 -486.7877} C_DIS
LIN {X -39.5245,Y -27.1169,Z 63,A -152.4255,B 24.8725,C -2.6057,E1 24.8669,E2 -483.9613} C_DIS
LIN {X -40.8075,Y -25.1448,Z 63,A -155.2545,B 24.8718,C -2.6126,E1 24.8627,E2 -481.1345} C_DIS
LIN {X -41.9921,Y -23.1122,Z 63,A -158.0839,B 24.8711,C -2.6198,E1 24.8588,E2 -478.3073} C_DIS
LIN {X -43.0756,Y -21.0239,Z 63,A -160.9138,B 24.8704,C -2.6271,E1 24.8553,E2 -475.4799} C_DIS
LIN {X -44.0553,Y -18.885,Z 63,A -163.7444,B 24.8697,C -2.6347,E1 24.852,E2 -472.6518} C_DIS
LIN {X -44.9289,Y -16.7005,Z 63,A -166.5754,B 24.8689,C -2.6425,E1 24.8492,E2 -469.8235} C_DIS
LIN {X -45.6387,Y -14.6474,Z 63,A -169.2097,B 24.8682,C -2.6496,E1 24.8469,E2 -467.1911} C_DIS
LIN {X -46.3495,Y -12.2163,Z 63,A -172.2384,B 24.8673,C -2.6585,E1 24.8446,E2 -464.1662} C_DIS
LIN {X -46.8931,Y -9.9273,Z 63,A -175.0705,B 24.8665,C -2.6667,E1 24.8429,E2 -461.3371} C_DIS
LIN {X -47.3237,Y -7.6145,Z 63,A -177.9028,B 24.8656,C -2.675,E1 24.8415,E2 -458.5079} C_DIS
LIN {X -47.6194,Y -5.4623,Z 63,A 179.4818,B 24.8648,C -2.6828,E1 24.8406,E2 -455.8954} C_DIS
LIN {X -47.83,Y -3.1192,Z 63,A 176.649,B 24.864,C -2.6913,E1 24.84,E2 -453.0659} C_DIS
LIN {X -47.9255,Y -0.7685,Z 63,A 173.7432,B 24.8632,C -2.6989,E1 24.8398,E2 -450.1608} C_DIS
LIN {X -47.8999,Y 1.7643,Z 63,A 170.7663,B 24.8622,C -2.7091,E1 24.84,E2 -447.1902} C_DIS
LIN {X -47.7556,Y 4.1125,Z 63,A 167.9333,B 24.8613,C -2.7176,E1 24.8405,E2 -444.3607} C_DIS
LIN {X -47.4963,Y 6.4508,Z 63,A 165.1005,B 24.8604,C -2.7262,E1 24.8415,E2 -441.5315} C_DIS
LIN {X -47.1545,Y 8.5961,Z 63,A 162.4849,B 24.8596,C -2.7341,E1 24.8427,E2 -438.9192} C_DIS
LIN {X -46.6714,Y 10.919,Z 63,A 159.5648,B 24.8588,C -2.7418,E1 24.8445,E2 -436.0004} C_DIS
LIN {X -46.0357,Y 13.3501,Z 63,A 156.6027,B 24.8578,C -2.7516,E1 24.8467,E2 -433.0444} C_DIS
LIN {X -45.3252,Y 15.5929,Z 63,A 153.7704,B 24.8569,C -2.7599,E1 24.8492,E2 -430.2158} C_DIS
LIN {X -44.5061,Y 17.7966,Z 63,A 150.94,B 24.8561,C -2.768,E1 24.852,E2 -427.389} C_DIS
LIN {X -43.5786,Y 19.9605,Z 63,A 148.1068,B 24.8552,C -2.7761,E1 24.8552,E2 -424.5595} C_DIS
LIN {X -42.5467,Y 22.0747,Z 63,A 145.2755,B 24.8544,C -2.784,E1 24.8588,E2 -421.7319} C_DIS
LIN {X -41.4123,Y 24.1358,Z 63,A 142.4449,B 24.8536,C -2.7917,E1 24.8626,E2 -418.9048} C_DIS
LIN {X -40.1781,Y 26.1387,Z 63,A 139.6145,B 24.8528,C -2.7992,E1 24.8669,E2 -416.078} C_DIS
LIN {X -38.8545,Y 28.0684,Z 63,A 136.7959,B 24.8521,C -2.8064,E1 24.8714,E2 -413.2628} C_DIS
LIN {X -37.4226,Y 29.951,Z 63,A 133.9552,B 24.8513,C -2.8135,E1 24.8763,E2 -410.4258} C_DIS
LIN {X -35.9079,Y 31.7512,Z 63,A 131.1265,B 24.8506,C -2.8203,E1 24.8814,E2 -407.6005} C_DIS
LIN {X -34.3067,Y 33.4748,Z 63,A 128.2984,B 24.8499,C -2.8269,E1 24.8868,E2 -404.7759} C_DIS
LIN {X -32.6228,Y 35.1179,Z 63,A 125.4711,B 24.8492,C -2.8332,E1 24.8926,E2 -401.9519} C_DIS
LIN {X -30.8604,Y 36.6763,Z 63,A 122.6443,B 24.8486,C -2.8392,E1 24.8985,E2 -399.1283} C_DIS
LIN {X -29.0236,Y 38.1464,Z 63,A 119.8183,B 24.848,C -2.8448,E1 24.9047,E2 -396.3055} C_DIS
LIN {X -27.1169,Y 39.5245,Z 63,A 116.9931,B 24.8474,C -2.8502,E1 24.9112,E2 -393.4833} C_DIS
LIN {X -25.1448,Y 40.8075,Z 63,A 114.1686,B 24.8468,C -2.8552,E1 24.9178,E2 -390.6618} C_DIS
LIN {X -23.1122,Y 41.9921,Z 63,A 111.345,B 24.8463,C -2.8598,E1 24.9247,E2 -387.841} C_DIS
LIN {X -21.0239,Y 43.0756,Z 63,A 108.5224,B 24.8459,C -2.8641,E1 24.9317,E2 -385.0212} C_DIS
LIN {X -18.885,Y 44.0553,Z 63,A 105.7003,B 24.8454,C -2.8681,E1 24.9389,E2 -382.2017} C_DIS
LIN {X -16.8045,Y 44.8895,Z 63,A 102.9723,B 24.8451,C -2.8709,E1 24.946,E2 -379.4746} C_DIS
LIN {X -14.4759,Y 45.6942,Z 63,A 100.0595,B 24.8447,C -2.8748,E1 24.9537,E2 -376.5657} C_DIS
LIN {X -12.2163,Y 46.3495,Z 63,A 97.2404,B 24.8444,C -2.8776,E1 24.9613,E2 -373.7488} C_DIS
LIN {X -9.9273,Y 46.8931,Z 63,A 94.4222,B 24.8442,C -2.88,E1 24.969,E2 -370.9326} C_DIS
LIN {X -7.7297,Y 47.3044,Z 63,A 91.702,B 24.844,C -2.8812,E1 24.9765,E2 -368.2127} C_DIS
LIN {X -5.2832,Y 47.6403,Z 63,A 88.7889,B 24.8438,C -2.8835,E1 24.9845,E2 -365.303} C_DIS
LIN {X -2.9392,Y 47.8422,Z 63,A 85.9735,B 24.8437,C -2.8846,E1 24.9923,E2 -362.4893} C_DIS
LIN {X -0.5882,Y 47.9288,Z 63,A 83.1593,B 24.8436,C -2.8854,E1 25.0002,E2 -359.6764} C_DIS
LIN {X 1.7643,Y 47.8999,Z 63,A 80.346,B 24.8436,C -2.8857,E1 25.0081,E2 -356.8644} C_DIS
LIN {X 4.1125,Y 47.7556,Z 63,A 77.5337,B 24.8436,C -2.8856,E1 25.0159,E2 -354.0532} C_DIS
LIN {X 6.4508,Y 47.4963,Z 63,A 74.7311,B 24.8436,C -2.8852,E1 25.0236,E2 -351.2518} C_DIS
LIN {X 8.7735,Y 47.1226,Z 63,A 71.9122,B 24.8437,C -2.8841,E1 25.0314,E2 -348.4334} C_DIS
LIN {X 11.0752,Y 46.6353,Z 63,A 69.1029,B 24.8439,C -2.8828,E1 25.0391,E2 -345.6246} C_DIS
LIN {X 13.3501,Y 46.0357,Z 63,A 66.2946,B 24.844,C -2.881,E1 25.0466,E2 -342.8167} C_DIS
LIN {X 15.5929,Y 45.3252,Z 63,A 63.4873,B 24.8443,C -2.8789,E1 25.0541,E2 -340.0097} C_DIS
LIN {X 17.7981,Y 44.5055,Z 63,A 60.681,B 24.8446,C -2.8763,E1 25.0614,E2 -337.2034} C_DIS
LIN {X 19.9605,Y 43.5786,Z 63,A 57.8753,B 24.8449,C -2.8733,E1 25.0685,E2 -334.3976} C_DIS
LIN {X 22.0747,Y 42.5467,Z 63,A 55.0709,B 24.8452,C -2.87,E1 25.0755,E2 -331.5929} C_DIS
LIN {X 24.1358,Y 41.4123,Z 63,A 52.2672,B 24.8456,C -2.8663,E1 25.0823,E2 -328.7887} C_DIS
LIN {X 26.1387,Y 40.1781,Z 63,A 49.4645,B 24.8461,C -2.8622,E1 25.089,E2 -325.9853} C_DIS
LIN {X 28.0787,Y 38.8472,Z 63,A 46.6624,B 24.8466,C -2.8578,E1 25.0954,E2 -323.1825} C_DIS
LIN {X 29.951,Y 37.4226,Z 63,A 43.8614,B 24.8471,C -2.853,E1 25.1015,E2 -320.3804} C_DIS
LIN {X 31.7512,Y 35.9079,Z 63,A 41.061,B 24.8476,C -2.8479,E1 25.1074,E2 -317.5788} C_DIS
LIN {X 33.4748,Y 34.3067,Z 63,A 38.2615,B 24.8482,C -2.8424,E1 25.1131,E2 -314.778} C_DIS
LIN {X 35.1179,Y 32.6228,Z 63,A 35.4627,B 24.8488,C -2.8367,E1 25.1185,E2 -311.9777} C_DIS
Enddeposition()
END
